FUNCTION_BLOCK "PRG_DSI_Status"
TITLE = Program Status DSI
{ S7_Optimized_Access := 'TRUE' }
AUTHOR : 'A.Schaefer'
VERSION : 0.0
   VAR
      lx_Init { ExternalAccessible := 'False'; ExternalVisible := 'False'; ExternalWritable := 'False'} : Bool;
      lx_Start { ExternalAccessible := 'False'; ExternalVisible := 'False'; ExternalWritable := 'False'} : Bool;
      li_StepCase { ExternalAccessible := 'False'; ExternalVisible := 'False'; ExternalWritable := 'False'} : Int;
      ldt_MQTT { ExternalAccessible := 'False'; ExternalVisible := 'False'; ExternalWritable := 'False'} : Date_And_Time;
      li_Return_LDT { ExternalAccessible := 'False'; ExternalVisible := 'False'; ExternalWritable := 'False'} : Int;
      lfb_R_Trig_Storage {InstructionName := 'R_TRIG'; LibVersion := '1.0'; ExternalAccessible := 'False'; ExternalVisible := 'False'; ExternalWritable := 'False'; S7_SetPoint := 'False'} : R_TRIG;
      lfb_F_Trig_Storage {InstructionName := 'F_TRIG'; LibVersion := '1.0'; ExternalAccessible := 'False'; ExternalVisible := 'False'; ExternalWritable := 'False'; S7_SetPoint := 'False'} : F_TRIG;
      lfb_TON_Status {InstructionName := 'TON_TIME'; LibVersion := '1.0'; ExternalAccessible := 'False'; ExternalVisible := 'False'; ExternalWritable := 'False'; S7_SetPoint := 'False'} : TON_TIME;
      lx_StartStatus { ExternalAccessible := 'False'; ExternalVisible := 'False'; ExternalWritable := 'False'} : Bool;
      lfb_TON_Schritt {InstructionName := 'TON_TIME'; LibVersion := '1.0'; ExternalAccessible := 'False'; ExternalVisible := 'False'; ExternalWritable := 'False'; S7_SetPoint := 'False'} : TON_TIME;
      lx_StartTimer { ExternalAccessible := 'False'; ExternalVisible := 'False'; ExternalWritable := 'False'} : Bool;
   END_VAR


BEGIN
	IF #lx_Init THEN

	    // wait time state
	    #lfb_TON_Status(IN := NOT #lx_StartStatus,
	                    PT := T#2s);

	    // rising/falling edge light barrier DSI
	    #lfb_R_Trig_Storage(CLK := NOT "IX_SSC_LightBarrierStorage_I3");
	    #lfb_F_Trig_Storage(CLK := NOT "IX_SSC_LightBarrierStorage_I3");

	    // state of the DSI transmitted to the cloud
	    IF (#lfb_TON_Status.Q OR #lfb_R_Trig_Storage.Q OR #lfb_F_Trig_Storage.Q) AND NOT #lx_StartStatus THEN
	        #lx_StartStatus := TRUE;
	        #li_Return_LDT := RD_SYS_T(#ldt_MQTT);
	        IF NOT "IX_SSC_LightBarrierStorage_I3" THEN
	            "gtyp_Interface_Dashboard".Subscribe.State_DSI.i_code := 0;
	            "gtyp_Interface_Dashboard".Subscribe.State_DSI.x_active := TRUE;
	        ELSE
	            "gtyp_Interface_Dashboard".Subscribe.State_DSI.i_code := 1;
	            IF #lfb_F_Trig_Storage.Q THEN
	                "gtyp_Interface_Dashboard".Subscribe.State_DSI.x_active := FALSE;
	            END_IF;
	        END_IF;
	        "gtyp_Interface_Dashboard".Subscribe.State_DSI.ldt_ts := DT_TO_LDT(#ldt_MQTT);
	        "gtyp_Interface_Dashboard".Subscribe.State_DSI.s_station := 'dsi';
	        "gtyp_Interface_Dashboard".Subscribe.State_DSI.s_target := '';
	        "gtyp_Interface_Dashboard".Subscribe.State_DSI.s_description := '';
	    END_IF;

	    IF NOT #lfb_TON_Status.Q AND #lx_StartStatus THEN
	        #lx_StartStatus := FALSE;
	    END_IF;
	ELSE
	    #lx_Init := TRUE;
	END_IF;
END_FUNCTION_BLOCK

FUNCTION_BLOCK "PRG_SLD_Ablauf"
TITLE = Program Ablauf SLD
{ S7_Optimized_Access := 'TRUE' }
AUTHOR : 'A.Schaefer'
VERSION : 0.0
   VAR
      lx_Init { ExternalAccessible := 'False'; ExternalVisible := 'False'; ExternalWritable := 'False'} : Bool;
      lx_Start_TON_Wait { ExternalAccessible := 'False'; ExternalVisible := 'False'; ExternalWritable := 'False'} : Bool;
      lx_Time_Error { ExternalAccessible := 'False'; ExternalVisible := 'False'; ExternalWritable := 'False'} : Bool;
      lt_TON_Wait { ExternalAccessible := 'False'; ExternalVisible := 'False'; ExternalWritable := 'False'} : Time;
      lx_Start_TON_State { ExternalAccessible := 'False'; ExternalVisible := 'False'; ExternalWritable := 'False'} : Bool;
      ldt_MQTT { ExternalAccessible := 'False'; ExternalVisible := 'False'; ExternalWritable := 'False'} : Date_And_Time;
      li_Return_LDT { ExternalAccessible := 'False'; ExternalVisible := 'False'; ExternalWritable := 'False'} : Int;
      li_Lights { ExternalAccessible := 'False'; ExternalVisible := 'False'; ExternalWritable := 'False'} : Int;
      li_Lights_old { ExternalAccessible := 'False'; ExternalVisible := 'False'; ExternalWritable := 'False'} : Int;
      lw_ColorValueMin { ExternalAccessible := 'False'; ExternalVisible := 'False'; ExternalWritable := 'False'} : Word;
      li_CounterActual { ExternalAccessible := 'False'; ExternalVisible := 'False'; ExternalWritable := 'False'} : Int;
      lx_White { ExternalAccessible := 'False'; ExternalVisible := 'False'; ExternalWritable := 'False'} : Bool;
      lx_Blue { ExternalAccessible := 'False'; ExternalVisible := 'False'; ExternalWritable := 'False'} : Bool;
      lx_Red { ExternalAccessible := 'False'; ExternalVisible := 'False'; ExternalWritable := 'False'} : Bool;
      li_StepCase { ExternalAccessible := 'False'; ExternalVisible := 'False'; ExternalWritable := 'False'} : Int;
      ls_Color { ExternalAccessible := 'False'; ExternalVisible := 'False'; ExternalWritable := 'False'} : String;
      lfb_TOF_ConveyerBelt_Out {InstructionName := 'TOF_TIME'; LibVersion := '1.0'; ExternalAccessible := 'False'; ExternalVisible := 'False'; ExternalWritable := 'False'; S7_SetPoint := 'False'} : TOF_TIME;
      lfb_TON_Wait {InstructionName := 'TON_TIME'; LibVersion := '1.0'; ExternalAccessible := 'False'; ExternalVisible := 'False'; ExternalWritable := 'False'; S7_SetPoint := 'False'} : TON_TIME;
      lfb_TON_Error {InstructionName := 'TON_TIME'; LibVersion := '1.0'; ExternalAccessible := 'False'; ExternalVisible := 'False'; ExternalWritable := 'False'; S7_SetPoint := 'False'} : TON_TIME;
      lfb_TON_State {InstructionName := 'TON_TIME'; LibVersion := '1.0'; ExternalAccessible := 'False'; ExternalVisible := 'False'; ExternalWritable := 'False'; S7_SetPoint := 'False'} : TON_TIME;
      lfb_F_Trig_Counter {InstructionName := 'F_TRIG'; LibVersion := '1.0'; ExternalAccessible := 'False'; ExternalVisible := 'False'; ExternalWritable := 'False'; S7_SetPoint := 'False'} : F_TRIG;
      lfb_R_Trig_Counter {InstructionName := 'R_TRIG'; LibVersion := '1.0'; ExternalAccessible := 'False'; ExternalVisible := 'False'; ExternalWritable := 'False'; S7_SetPoint := 'False'} : R_TRIG;
   END_VAR


BEGIN
	IF #lx_Init THEN

	    // Restart after set Positioning
	    IF "gtyp_Setup".x_Color_Sensor_Calibration THEN
	        #li_StepCase := 0;
	    END_IF;

	    // wait time state
	    #lfb_TON_State(IN := NOT #lx_Start_TON_State,
	                    PT := T#2s);

	    // state of the SLD cyclically transmitted to the cloud
	    IF (#lfb_TON_State.Q OR (#li_Lights <> #li_Lights_old)) AND NOT #lx_Start_TON_State THEN
	        #li_Lights_old := #li_Lights;
	        #lx_Start_TON_State := TRUE;
	        #li_Return_LDT := RD_SYS_T(#ldt_MQTT);
	        "gtyp_Interface_Dashboard".Subscribe.State_SLD.ldt_ts := DT_TO_LDT(#ldt_MQTT);
	        "gtyp_Interface_Dashboard".Subscribe.State_SLD.i_code := #li_Lights;
	        "gtyp_Interface_Dashboard".Subscribe.State_SLD.s_description := '';
	        "gtyp_Interface_Dashboard".Subscribe.State_SLD.s_station := 'sld';
	        "gtyp_Interface_Dashboard".Subscribe.State_SLD.s_target := '';
	    END_IF;

	    // restart wait time state
	    IF NOT #lfb_TON_State.Q AND #lx_Start_TON_State THEN
	        #lx_Start_TON_State := FALSE;
	    END_IF;

	    // FB TON Wait
	    #lfb_TON_Wait(IN := #lx_Start_TON_Wait,
	                     PT := #lt_TON_Wait);

	    // runtime monitoring error
	    #lfb_TON_Error(IN:= #lx_Time_Error,
	                   PT:= T#30s);

	    // rising edge pulse counter
	    #lfb_R_Trig_Counter(CLK:= "IX_SLD_PulseCounter_I1");

	    // falling edge pulse counter
	    #lfb_F_Trig_Counter(CLK := "IX_SLD_PulseCounter_I1");

	    // step chain SLD
	    CASE #li_StepCase OF

	        0:  // Init
	            #lx_Start_TON_Wait := FALSE;
	            #lx_Time_Error := FALSE;
	            #li_Lights := 1;

	            IF NOT "gtyp_SLD".x_Error AND NOT "gtyp_Setup".x_Color_Sensor_Calibration THEN
	                #li_StepCase := 10;
	            END_IF;

	        10: // turn-on Compressor and wait sequence
	            #li_Lights := 2;
	            "QX_SLD_Compressor_Q2" := TRUE;

	            #lx_Start_TON_Wait := TRUE;
	            #lt_TON_Wait := T#1000ms;

	            IF #lfb_TON_Wait.Q THEN
	                #lx_Start_TON_Wait := FALSE;
	                #li_StepCase := 20;
	            END_IF;

	        20:  // reset Ejectors
	            "QX_SLD_ValveFirstEjectorWhite_Q3"  := FALSE;
	            "QX_SLD_ValveSecondEjectorRed_Q4"   := FALSE;
	            "QX_SLD_ValveThirdEjectorBlue_Q5"   := FALSE;
	            "QX_SLD_M1_ConveyorBelt_Q1"         := FALSE;

	            #lx_Start_TON_Wait := TRUE;
	            #lt_TON_Wait := T#2000ms;

	            IF #lfb_TON_Wait.Q THEN
	                #lx_Start_TON_Wait := FALSE;
	                #li_StepCase := 30;
	            END_IF;

	        30: // turn-off Compressor

	            "QX_SLD_Compressor_Q2" := FALSE;

	            #li_StepCase := 40;

	        40: // start belt if Light barrier I2 active

	            #li_Lights := 1;
	            IF NOT "IX_SLD_LightBarrierInlet_I2" THEN
	                "gtyp_Interface_Dashboard".Subscribe.State_SLD.x_active := TRUE;
	                #li_Lights := 2;
	                "QX_SLD_Compressor_Q2"      := TRUE;
	                "QX_SLD_M1_ConveyorBelt_Q1" := TRUE;
	                #lw_ColorValueMin           := 40000;
	                #li_CounterActual := 0;
	                #lx_Blue := FALSE;
	                #lx_Red := FALSE;
	                #lx_White := FALSE;
	                #li_StepCase := 50;
	            END_IF;

	        50: // take the min Value of the Color sensor
	            IF #lw_ColorValueMin > "IW_SLD_ColorSensor_A4" THEN
	                #lw_ColorValueMin := "IW_SLD_ColorSensor_A4";
	            END_IF;

	            #lx_Time_Error := TRUE;

	            // Stop when light barrier I3 on
	            IF NOT "IX_SLD_LightBarrierBehindColorSensor_I3" THEN
	                #lx_Time_Error  := FALSE;
	                #li_StepCase    := 60;
	            END_IF;

	            // runtime error
	            IF #lfb_TON_Error.Q THEN
	                #li_Lights                  := 4;
	                #lx_Time_Error              := FALSE;
	                "QX_SLD_Compressor_Q2"      := FALSE;
	                "QX_SLD_M1_ConveyorBelt_Q1" := FALSE;
	                "gtyp_Interface_Dashboard".Subscribe.State_SLD.x_active := FALSE;
	                "gtyp_SLD".x_Error          := TRUE;
	                #li_StepCase                := 0;
	            END_IF;

	        60: // analyze color

	            IF #lw_ColorValueMin >= "gtyp_SLD".w_Threshold_Red_Blue THEN
	                #lx_Blue := TRUE;
	            ELSIF #lw_ColorValueMin <= "gtyp_SLD".w_Threshold_White_Red THEN
	                #lx_White := TRUE;
	            ELSIF #lw_ColorValueMin > "gtyp_SLD".w_Threshold_White_Red AND #lw_ColorValueMin < "gtyp_SLD".w_Threshold_Red_Blue THEN
	                #lx_Red := TRUE;
	            END_IF;

	            // actual counter
	            IF #lfb_R_Trig_Counter.Q OR #lfb_F_Trig_Counter.Q THEN
	                #li_CounterActual := #li_CounterActual + 1;
	            END_IF;

	            // Reached counter value and color set Ejector
	            IF (#li_CounterActual = "gtyp_SLD".i_CounterValue_Blue) AND #lx_Blue THEN
	                "QX_SLD_ValveThirdEjectorBlue_Q5" := TRUE;
	                #li_Return_LDT := RD_SYS_T(#ldt_MQTT);
	                "gtyp_SLD".Workpiece.s_state := 'PROCESSED';
	                "gtyp_SLD".History[7].i_code := 700;
	                "gtyp_SLD".History[7].ldt_ts := DT_TO_LDT(#ldt_MQTT);
	                #li_StepCase := 70;
	            ELSIF (#li_CounterActual = "gtyp_SLD".i_CounterValue_White) AND #lx_White THEN
	                "QX_SLD_ValveFirstEjectorWhite_Q3" := TRUE;
	                #li_Return_LDT := RD_SYS_T(#ldt_MQTT);
	                "gtyp_SLD".Workpiece.s_state := 'PROCESSED';
	                "gtyp_SLD".History[7].i_code := 700;
	                "gtyp_SLD".History[7].ldt_ts := DT_TO_LDT(#ldt_MQTT);
	                #li_StepCase := 70;
	            ELSIF (#li_CounterActual = "gtyp_SLD".i_CounterValue_Red) AND #lx_Red THEN
	                "QX_SLD_ValveSecondEjectorRed_Q4" := TRUE;
	                #li_Return_LDT := RD_SYS_T(#ldt_MQTT);
	                "gtyp_SLD".Workpiece.s_state := 'PROCESSED';
	                "gtyp_SLD".History[7].i_code := 700;
	                "gtyp_SLD".History[7].ldt_ts := DT_TO_LDT(#ldt_MQTT);
	                #li_StepCase := 70;
	            ELSIF (#li_CounterActual = 80) THEN
	                #li_Lights := 4;
	                "gtyp_SLD".x_Error := TRUE;
	                #li_StepCase := 70;
	            END_IF;

	        70: // wait sequence
	            #lx_Start_TON_Wait := TRUE;
	            #lt_TON_Wait := T#500ms;

	            IF #lfb_TON_Wait.Q THEN
	                "QX_SLD_ValveThirdEjectorBlue_Q5" := FALSE;
	                "QX_SLD_ValveFirstEjectorWhite_Q3" := FALSE;
	                "QX_SLD_ValveSecondEjectorRed_Q4" := FALSE;
	                #lx_Start_TON_Wait := FALSE;
	                #li_StepCase := 80;
	            END_IF;

	        80: // wait sequence

	            #lx_Start_TON_Wait := TRUE;
	            #lt_TON_Wait := T#2000ms;

	            IF #lfb_TON_Wait.Q THEN
	                "QX_SLD_Compressor_Q2" := FALSE;
	                #lx_Start_TON_Wait := FALSE;
	                #li_StepCase := 90;
	            END_IF;

	        90: // Stop belt
	            "QX_SLD_M1_ConveyorBelt_Q1"    := FALSE;
	            #li_StepCase := 40;
	        // Statement section ELSE
	        ELSE
	            ;
	    END_CASE;

	ELSE
	    "gtyp_SLD".x_Error := FALSE;
	    #li_Lights := 1;
	    #lx_Init := TRUE;
	END_IF;
END_FUNCTION_BLOCK

FUNCTION_BLOCK "PRG_HBW_Axis_Horizontal"
TITLE = Program Axis horizontal HBW
{ S7_Optimized_Access := 'TRUE' }
AUTHOR : 'A.Schaefer'
VERSION : 0.0
   VAR
      lx_Init { ExternalAccessible := 'False'; ExternalVisible := 'False'; ExternalWritable := 'False'} : Bool;
      lfb_Horizontal_Axis { ExternalAccessible := 'False'; ExternalVisible := 'False'; ExternalWritable := 'False'; S7_SetPoint := 'False'} : "FB_Axis";
   END_VAR


BEGIN
	IF #lx_Init THEN

	    // FB Axis horizontal
	    #lfb_Horizontal_Axis(ini_Axis               := 6,
	                         indi_Increment          := "gtyp_HBW".Horizontal_Axis.di_Increment,
	                         inx_Ref_Switch         := "IX_HBW_RefSwitchHorizontalAxis_I1",
	                         inx_Referencing        := "gtyp_HBW".Horizontal_Axis.x_Reference,
	                         inx_Start_Positioning  := "gtyp_HBW".Horizontal_Axis.x_Start_Positioning,
	                         indi_Target_Position   := "gtyp_HBW".Horizontal_Axis.di_Target_Position,
	                         ini_PWM                := "gtyp_HBW".Horizontal_Axis.i_PWM,
	                         inouttyp_Config        := "gtyp_HBW".Horizontal_Axis.Config,
	                         inouttyp_Setup         := "gtyp_SetupAxis");

	    "QX_HBW_M2_HorizontalTowardsRack_Q3"            := #lfb_Horizontal_Axis.outx_Motor_Pos;
	    "QX_HBW_M2_HorizontalTowardsConveyorBelt_Q4"    := #lfb_Horizontal_Axis.outx_Motor_Neg;
	    "QW_HBW_PWM_HorizontalAxis_M2"                  := #lfb_Horizontal_Axis.outi_Motor_PWM;
	    "gtyp_HBW".Horizontal_Axis.di_Actual_Position   := #lfb_Horizontal_Axis.outdi_Actual_Position;
	    "gtyp_HBW".Horizontal_Axis.x_Referenced         := #lfb_Horizontal_Axis.outx_Referenced;
	    "gtyp_HBW".Horizontal_Axis.x_Position_Reached   := #lfb_Horizontal_Axis.outx_Position_Reached;
	ELSE
	    #lx_Init := TRUE;
	END_IF;
END_FUNCTION_BLOCK

FUNCTION_BLOCK "PRG_SSC_Light"
TITLE = Program Lights
{ S7_Optimized_Access := 'TRUE' }
AUTHOR : 'A.Schaefer'
VERSION : 0.0
   VAR
      lx_Init { ExternalAccessible := 'False'; ExternalVisible := 'False'; ExternalWritable := 'False'} : Bool;
      lx_Start { ExternalAccessible := 'False'; ExternalVisible := 'False'; ExternalWritable := 'False'} : Bool;
      li_StepCase { ExternalAccessible := 'False'; ExternalVisible := 'False'; ExternalWritable := 'False'} : Int;
      ldt_MQTT { ExternalAccessible := 'False'; ExternalVisible := 'False'; ExternalWritable := 'False'} : Date_And_Time;
      lldt_ts_old { ExternalAccessible := 'False'; ExternalVisible := 'False'; ExternalWritable := 'False'} : LDT;
      li_Return_LDT { ExternalAccessible := 'False'; ExternalVisible := 'False'; ExternalWritable := 'False'} : Int;
      lfb_TOF_Camera {InstructionName := 'TOF_TIME'; LibVersion := '1.0'; ExternalAccessible := 'False'; ExternalVisible := 'False'; ExternalWritable := 'False'; S7_SetPoint := 'False'} : TOF_TIME;
      lfb_TON_Schritt {InstructionName := 'TON_TIME'; LibVersion := '1.0'; ExternalAccessible := 'False'; ExternalVisible := 'False'; ExternalWritable := 'False'; S7_SetPoint := 'False'} : TON_TIME;
      lfb_blinker_cam { ExternalAccessible := 'False'; ExternalVisible := 'False'; ExternalWritable := 'False'; S7_SetPoint := 'False'} : "FB_Blinker";
      lfb_blinker_config { ExternalAccessible := 'False'; ExternalVisible := 'False'; ExternalWritable := 'False'; S7_SetPoint := 'False'} : "FB_Blinker";
      lx_StartTimer { ExternalAccessible := 'False'; ExternalVisible := 'False'; ExternalWritable := 'False'} : Bool;
   END_VAR


BEGIN
	IF #lx_Init THEN

	    // if camera sen picture - Red light flash
	    IF "gtyp_Interface_Dashboard".Subscribe.CameraPicture.ldt_ts > #lldt_ts_old THEN
	        #lldt_ts_old := "gtyp_Interface_Dashboard".Subscribe.CameraPicture.ldt_ts;
	        #lfb_blinker_cam(int_periodendauer := T#50ms);
	    END_IF;

	    // reload flash
	    "QX_SSC_LED_Red_Online_Q8":= #lfb_blinker_cam.outx_blinker;

	    // FB flash config
	    #lfb_blinker_config(int_periodendauer := T#500ms);

	    //  Deciding which state
	    //  Setup - Calibration State
	    IF "gtyp_Setup".x_Set_Pos_Activ OR "gtyp_Setup".x_Color_Sensor_Calibration
	                                    OR "gtyp_Setup".x_Counter_Value_Calibration
	                                    OR "gtyp_Setup".x_Clean_Rack_HBW THEN
	        "QX_SSC_LED_Green_Q5"  := #lfb_blinker_config.outx_blinker;
	        "QX_SSC_LED_Yellow_Q6" := #lfb_blinker_config.outx_blinker;
	        "QX_SSC_LED_Red_Q7"    := #lfb_blinker_config.outx_blinker;
	    //  Error State
	    ELSIF ("gtyp_Interface_Dashboard".Subscribe.State_HBW.i_code = 4)
	        OR ("gtyp_Interface_Dashboard".Subscribe.State_MPO.i_code = 4)
	        OR ("gtyp_Interface_Dashboard".Subscribe.State_SLD.i_code = 4)
	        OR ("gtyp_Interface_Dashboard".Subscribe.State_VGR.i_code = 4) THEN
	        "QX_SSC_LED_Green_Q5" := FALSE;
	        "QX_SSC_LED_Yellow_Q6" := FALSE;
	        "QX_SSC_LED_Red_Q7" := TRUE;
	    //  Proccessing State
	    ELSIF ("gtyp_Interface_Dashboard".Subscribe.State_HBW.i_code = 2)
	        OR ("gtyp_Interface_Dashboard".Subscribe.State_MPO.i_code = 2)
	        OR ("gtyp_Interface_Dashboard".Subscribe.State_SLD.i_code = 2)
	        OR ("gtyp_Interface_Dashboard".Subscribe.State_VGR.i_code = 2) THEN
	            "QX_SSC_LED_Green_Q5" := FALSE;
	            "QX_SSC_LED_Yellow_Q6" := TRUE;
	            "QX_SSC_LED_Red_Q7" := FALSE;
	    //  Idle State
	    ELSIF ("gtyp_Interface_Dashboard".Subscribe.State_HBW.i_code = 1)
	        AND ("gtyp_Interface_Dashboard".Subscribe.State_MPO.i_code = 1)
	        AND ("gtyp_Interface_Dashboard".Subscribe.State_SLD.i_code = 1)
	        AND ("gtyp_Interface_Dashboard".Subscribe.State_VGR.i_code = 1) THEN
	            "QX_SSC_LED_Green_Q5" := TRUE;
	            "QX_SSC_LED_Yellow_Q6" := FALSE;
	            "QX_SSC_LED_Red_Q7" := FALSE;
	    //  nothing State
	    ELSE
	        "QX_SSC_LED_Green_Q5" := FALSE;
	        "QX_SSC_LED_Yellow_Q6" := FALSE;
	        "QX_SSC_LED_Red_Q7" := FALSE;
	    END_IF;


	ELSE
	    #lx_Init := TRUE;
	END_IF;
END_FUNCTION_BLOCK

FUNCTION_BLOCK "PRG_DSO_Status"
TITLE = Program Status DSO
{ S7_Optimized_Access := 'TRUE' }
AUTHOR : 'A.Schaefer'
VERSION : 0.0
   VAR
      lx_Init { ExternalAccessible := 'False'; ExternalVisible := 'False'; ExternalWritable := 'False'} : Bool;
      lx_Start { ExternalAccessible := 'False'; ExternalVisible := 'False'; ExternalWritable := 'False'} : Bool;
      li_StepCase { ExternalAccessible := 'False'; ExternalVisible := 'False'; ExternalWritable := 'False'} : Int;
      ldt_MQTT { ExternalAccessible := 'False'; ExternalVisible := 'False'; ExternalWritable := 'False'} : Date_And_Time;
      li_Return_LDT { ExternalAccessible := 'False'; ExternalVisible := 'False'; ExternalWritable := 'False'} : Int;
      li_code_old { ExternalAccessible := 'False'; ExternalVisible := 'False'; ExternalWritable := 'False'} : Int;
      lfb_R_Trig_Outsourcing {InstructionName := 'R_TRIG'; LibVersion := '1.0'; ExternalAccessible := 'False'; ExternalVisible := 'False'; ExternalWritable := 'False'; S7_SetPoint := 'False'} : R_TRIG;
      lfb_R_Trig_Take_Workpiece {InstructionName := 'R_TRIG'; LibVersion := '1.0'; ExternalAccessible := 'False'; ExternalVisible := 'False'; ExternalWritable := 'False'; S7_SetPoint := 'False'} : R_TRIG;
      lfb_TON_Status {InstructionName := 'TON_TIME'; LibVersion := '1.0'; ExternalAccessible := 'False'; ExternalVisible := 'False'; ExternalWritable := 'False'; S7_SetPoint := 'False'} : TON_TIME;
      lfb_TON_End_Order {InstructionName := 'TON_TIME'; LibVersion := '1.0'; ExternalAccessible := 'False'; ExternalVisible := 'False'; ExternalWritable := 'False'; S7_SetPoint := 'False'} : TON_TIME;
      lx_StartStatus { ExternalAccessible := 'False'; ExternalVisible := 'False'; ExternalWritable := 'False'} : Bool;
      lx_StartEndOrder { ExternalAccessible := 'False'; ExternalVisible := 'False'; ExternalWritable := 'False'} : Bool;
      lx_StartTimer { ExternalAccessible := 'False'; ExternalVisible := 'False'; ExternalWritable := 'False'} : Bool;
   END_VAR


BEGIN
	IF #lx_Init THEN

	    // wait time state
	    #lfb_TON_Status(IN := NOT #lx_StartStatus,
	                    PT := T#2s);

	    // rising/falling edge light barrier DSI
	    #lfb_R_Trig_Outsourcing(CLK := NOT "IX_SSC_LightBarrierOutsourcing_I4");
	    #lfb_R_Trig_Take_Workpiece(CLK := "IX_SSC_LightBarrierOutsourcing_I4");

	    // start wait time end order
	    IF NOT "IX_SSC_LightBarrierOutsourcing_I4" AND ("gtyp_Interface_Dashboard".Subscribe.State_Order.s_state = 'SHIPPED') THEN
	        #lx_StartEndOrder := TRUE;
	    END_IF;

	    // wait time end order
	    #lfb_TON_End_Order(IN := #lx_StartEndOrder,
	                       PT := T#5s);

	    IF #lfb_R_Trig_Take_Workpiece.Q OR #lfb_TON_End_Order.Q THEN
	        #lx_StartEndOrder := FALSE;
	        "gtyp_Interface_Dashboard".Subscribe.State_Order.ldt_ts := DT_TO_LDT(#ldt_MQTT);
	        "gtyp_Interface_Dashboard".Subscribe.State_Order.s_state := 'WAITING_FOR_ORDER';
	        "gtyp_Interface_Dashboard".Subscribe.State_Order.s_type := '';
	        "gtyp_Interface_Dashboard".Subscribe.State_DSO.x_active := FALSE;
	    END_IF;

	    // state of the DSO transmitted to the cloud
	    IF (#lfb_TON_Status.Q OR #lfb_R_Trig_Outsourcing.Q OR #lfb_R_Trig_Take_Workpiece.Q) AND NOT #lx_StartStatus THEN
	        #lx_StartStatus := TRUE;
	        #li_Return_LDT := RD_SYS_T(#ldt_MQTT);
	        IF NOT "IX_SSC_LightBarrierOutsourcing_I4" THEN
	            "gtyp_Interface_Dashboard".Subscribe.State_DSO.i_code := 0;
	        ELSE
	            "gtyp_Interface_Dashboard".Subscribe.State_DSO.i_code := 1;
	        END_IF;
	        "gtyp_Interface_Dashboard".Subscribe.State_DSO.ldt_ts := DT_TO_LDT(#ldt_MQTT);
	        "gtyp_Interface_Dashboard".Subscribe.State_DSO.s_station := 'dso';
	        "gtyp_Interface_Dashboard".Subscribe.State_DSO.s_target := '';
	        "gtyp_Interface_Dashboard".Subscribe.State_DSO.s_description := '';
	    END_IF;

	    IF NOT #lfb_TON_Status.Q AND #lx_StartStatus THEN
	        #lx_StartStatus := FALSE;
	    END_IF;
	ELSE
	    #lx_Init := TRUE;
	    #lx_StartEndOrder := FALSE;
	END_IF;
END_FUNCTION_BLOCK

FUNCTION_BLOCK "PRG_SSC_Set_Positioning"
TITLE = Program Set Positioning SSC
{ S7_Optimized_Access := 'TRUE' }
AUTHOR : 'A.Schaefer'
VERSION : 0.0
   VAR
      lx_Init { ExternalAccessible := 'False'; ExternalVisible := 'False'; ExternalWritable := 'False'} : Bool;
      lx_Start_TON_Wait { ExternalAccessible := 'False'; ExternalVisible := 'False'; ExternalWritable := 'False'} : Bool;
      lx_Start_Positioning_m { ExternalAccessible := 'False'; ExternalVisible := 'False'; ExternalWritable := 'False'} : Bool;
      lt_TON_Wait { ExternalAccessible := 'False'; ExternalVisible := 'False'; ExternalWritable := 'False'} : Time;
      li_StepCase { ExternalAccessible := 'False'; ExternalVisible := 'False'; ExternalWritable := 'False'} : Int;
      ldi_Pos_Horizontal { ExternalAccessible := 'False'; ExternalVisible := 'False'; ExternalWritable := 'False'} : DInt;
      ldi_Pos_Vertical { ExternalAccessible := 'False'; ExternalVisible := 'False'; ExternalWritable := 'False'} : DInt;
      lfb_R_Trig_Deaktivate {InstructionName := 'R_TRIG'; LibVersion := '1.0'; ExternalAccessible := 'False'; ExternalVisible := 'False'; ExternalWritable := 'False'; S7_SetPoint := 'False'} : R_TRIG;
      lfb_TON_Wait {InstructionName := 'TON_TIME'; LibVersion := '1.0'; ExternalAccessible := 'False'; ExternalVisible := 'False'; ExternalWritable := 'False'; S7_SetPoint := 'False'} : TON_TIME;
   END_VAR


BEGIN
	IF #lx_Init THEN

	    // FB TON Wait
	    #lfb_TON_Wait(IN := #lx_Start_TON_Wait,
	                  PT := #lt_TON_Wait);

	    #lfb_R_Trig_Deaktivate(CLK:= NOT "gtyp_Setup".x_Set_Pos_Activ
	                           OR NOT (("gtyp_Setup".i_Pos_Selection > 0)
	                           AND ("gtyp_Setup".i_Pos_Selection < 21)));
	    // Deaktivate step 10
	    IF #lfb_R_Trig_Deaktivate.Q THEN
	        "gtyp_SSC".Horizontal_Axis.x_Start_Positioning := FALSE;
	        "gtyp_SSC".Vertical_Axis.x_Start_Positioning := FALSE;
	        "gtyp_SSC".Horizontal_Axis.x_Reference := FALSE;
	        "gtyp_SSC".Vertical_Axis.x_Reference := FALSE;
	        "gtyp_Setup".x_Start_Positioning := FALSE;
	        "gtyp_Setup".x_Final_Positioning := FALSE;
	        "gtyp_Setup".x_Home_Positioning := FALSE;
	        "gtyp_Setup".x_Start_Offset := FALSE;
	        #lx_Start_Positioning_m := FALSE;
	        IF (#li_StepCase > 10) THEN
	            #li_StepCase            := 70;
	        END_IF;
	    END_IF;

	    // Set Positioning activ?
	    IF "gtyp_Setup".x_Set_Pos_Activ
	        AND (("gtyp_Setup".i_Pos_Selection > 0)
	        AND ("gtyp_Setup".i_Pos_Selection < 21))
	        AND ((#li_StepCase = 40)
	        OR (#li_StepCase = 60)) THEN

	        // Deciding which Position
	        // Position - Centre
	        IF "gtyp_Setup".i_Pos_Selection = 1 THEN
	            #ldi_Pos_Horizontal := "gtyp_SSC".di_Pos_Centre_Horizontal;
	            #ldi_Pos_Vertical := "gtyp_SSC".di_Pos_Centre_Vertical;
	            // Position - HBW
	        ELSIF "gtyp_Setup".i_Pos_Selection = 2 THEN
	            #ldi_Pos_Horizontal := "gtyp_SSC".di_Pos_HBW_Horizontal;
	            #ldi_Pos_Vertical := "gtyp_SSC".di_Pos_HBW_Vertical;
	        END_IF;
	    END_IF;

	    // Set Positioning activ?
	    IF NOT "gtyp_Setup".x_Set_Pos_Activ THEN
	        "gtyp_Setup".i_Pos_Selection := 0;
	    END_IF;

	    // step chain HBW
	    CASE #li_StepCase OF

	        0:  // init
	            #lx_Start_TON_Wait := FALSE;
	            #li_StepCase := 10;

	        10:  // Set Positioning activ?
	            IF "gtyp_Setup".x_Set_Pos_Activ
	                AND (("gtyp_Setup".i_Pos_Selection > 0)
	                AND ("gtyp_Setup".i_Pos_Selection < 21)) THEN
	                "gtyp_SSC".Horizontal_Axis.x_Start_Positioning := FALSE;
	                "gtyp_SSC".Vertical_Axis.x_Start_Positioning := FALSE;
	                "gtyp_SSC".Horizontal_Axis.x_Reference := FALSE;
	                "gtyp_SSC".Vertical_Axis.x_Reference := FALSE;
	                "gtyp_Setup".x_Start_Positioning := FALSE;
	                "gtyp_Setup".x_Final_Positioning := FALSE;
	                "gtyp_Setup".x_Home_Positioning  := FALSE;
	                "gtyp_Setup".x_Start_Offset := FALSE;
	                #li_StepCase := 20;
	            END_IF;

	        20: //homing vertical/horizontal axis

	            "gtyp_SSC".Horizontal_Axis.x_Reference := TRUE;
	            "gtyp_SSC".Vertical_Axis.x_Reference := TRUE;

	            IF NOT "gtyp_SSC".Horizontal_Axis.x_Referenced AND NOT "gtyp_SSC".Vertical_Axis.x_Referenced THEN
	                #li_StepCase := 30;
	            END_IF;

	        30: // homed vertical/horizontal axis
	            IF "gtyp_SSC".Horizontal_Axis.x_Referenced THEN
	                "gtyp_SSC".Horizontal_Axis.x_Reference := FALSE;
	            END_IF;
	            IF "gtyp_SSC".Vertical_Axis.x_Referenced THEN
	                "gtyp_SSC".Vertical_Axis.x_Reference := FALSE;
	            END_IF;

	            IF "gtyp_SSC".Horizontal_Axis.x_Referenced AND "gtyp_SSC".Vertical_Axis.x_Referenced THEN
	                "gtyp_SSC".Horizontal_Axis.x_Reference := FALSE;
	                "gtyp_SSC".Vertical_Axis.x_Reference := FALSE;
	                #li_StepCase := 40;
	            END_IF;

	        40:  // Start Positioning Step next
	            IF "gtyp_Setup".x_Start_Positioning OR #lx_Start_Positioning_m THEN
	                #lx_Start_Positioning_m := FALSE;
	                #li_StepCase            := 50;
	            END_IF;

	        50: // Position vertical/horizontal HBW
	            "gtyp_SSC".Horizontal_Axis.di_Target_Position := #ldi_Pos_Horizontal;
	            "gtyp_SSC".Horizontal_Axis.x_Start_Positioning := TRUE;
	            "gtyp_SSC".Vertical_Axis.di_Target_Position := #ldi_Pos_Vertical;
	            "gtyp_SSC".Vertical_Axis.x_Start_Positioning := TRUE;

	            IF ("gtyp_SSC".Horizontal_Axis.di_Actual_Position <= (#ldi_Pos_Horizontal + "gtyp_SSC".Horizontal_Axis.Config.di_Pos_Window))
	                AND ("gtyp_SSC".Horizontal_Axis.di_Actual_Position >= (#ldi_Pos_Horizontal - "gtyp_SSC".Horizontal_Axis.Config.di_Pos_Window))
	                AND "gtyp_SSC".Horizontal_Axis.x_Position_Reached THEN
	                "gtyp_SSC".Horizontal_Axis.x_Start_Positioning := FALSE;
	            END_IF;

	            IF ("gtyp_SSC".Vertical_Axis.di_Actual_Position <= (#ldi_Pos_Vertical + "gtyp_SSC".Vertical_Axis.Config.di_Pos_Window))
	                AND ("gtyp_SSC".Vertical_Axis.di_Actual_Position >= (#ldi_Pos_Vertical - "gtyp_SSC".Vertical_Axis.Config.di_Pos_Window))
	                AND "gtyp_SSC".Vertical_Axis.x_Position_Reached THEN
	                "gtyp_SSC".Vertical_Axis.x_Start_Positioning := FALSE;
	            END_IF;

	            IF ("gtyp_SSC".Horizontal_Axis.di_Actual_Position <= (#ldi_Pos_Horizontal + "gtyp_SSC".Horizontal_Axis.Config.di_Pos_Window))
	                AND ("gtyp_SSC".Horizontal_Axis.di_Actual_Position >= (#ldi_Pos_Horizontal - "gtyp_SSC".Horizontal_Axis.Config.di_Pos_Window))
	                AND "gtyp_SSC".Horizontal_Axis.x_Position_Reached
	                AND ("gtyp_SSC".Vertical_Axis.di_Actual_Position <= (#ldi_Pos_Vertical + "gtyp_SSC".Vertical_Axis.Config.di_Pos_Window))
	                AND ("gtyp_SSC".Vertical_Axis.di_Actual_Position >= (#ldi_Pos_Vertical - "gtyp_SSC".Vertical_Axis.Config.di_Pos_Window))
	                AND "gtyp_SSC".Vertical_Axis.x_Position_Reached THEN
	                "gtyp_SSC".Horizontal_Axis.x_Start_Positioning := FALSE;
	                "gtyp_SSC".Vertical_Axis.x_Start_Positioning := FALSE;
	                "gtyp_Setup".x_Start_Positioning := FALSE;
	                #li_StepCase := 60;
	            END_IF;

	        60: // Deciding which doing

	            // Start new Positioning
	            IF "gtyp_Setup".x_Start_Positioning OR "gtyp_Setup".x_Home_Positioning THEN
	                #lx_Start_Positioning_m := TRUE;
	                #li_StepCase            := 10;
	            ELSIF #lfb_R_Trig_Deaktivate.Q THEN
	                "gtyp_Setup".x_Home_Positioning := FALSE;
	                #li_StepCase                    := 70;
	            END_IF;

	        70: //homing vertical/horizontal axis

	            "gtyp_SSC".Horizontal_Axis.x_Reference := TRUE;
	            "gtyp_SSC".Vertical_Axis.x_Reference := TRUE;

	            IF NOT "gtyp_SSC".Horizontal_Axis.x_Referenced AND NOT "gtyp_SSC".Vertical_Axis.x_Referenced THEN
	                #li_StepCase := 80;
	            END_IF;

	        80: // homed vertical/horizontal axis
	            IF "gtyp_SSC".Horizontal_Axis.x_Referenced THEN
	                "gtyp_SSC".Horizontal_Axis.x_Reference := FALSE;
	            END_IF;
	            IF "gtyp_SSC".Vertical_Axis.x_Referenced THEN
	                "gtyp_SSC".Vertical_Axis.x_Reference := FALSE;
	            END_IF;

	            IF "gtyp_SSC".Horizontal_Axis.x_Referenced AND "gtyp_SSC".Vertical_Axis.x_Referenced THEN
	                "gtyp_SSC".Horizontal_Axis.x_Reference := FALSE;
	                "gtyp_SSC".Vertical_Axis.x_Reference := FALSE;
	                #li_StepCase := 0;
	            END_IF;

	            // Statement section ELSE
	        ELSE
	            ;
	    END_CASE;

	    IF (("gtyp_Setup".i_Pos_Selection > 0)
	        AND ("gtyp_Setup".i_Pos_Selection < 21)) THEN
	        // Reload Pos Value
	        "gtyp_Setup".di_Pos_Horizontal := #ldi_Pos_Horizontal;
	        "gtyp_Setup".di_Pos_Vertical := #ldi_Pos_Vertical;
	        "gtyp_Setup".di_Pos_Rotate := 0;
	    END_IF;
	ELSE
	    #lx_Init := TRUE;
	END_IF;
END_FUNCTION_BLOCK

FUNCTION_BLOCK "PRG_HBW_Set_Positioning"
TITLE = Program Set Positioning HBW
{ S7_Optimized_Access := 'TRUE' }
AUTHOR : 'A.Schaefer'
VERSION : 0.0
   VAR
      lx_Init { ExternalAccessible := 'False'; ExternalVisible := 'False'; ExternalWritable := 'False'} : Bool;
      lx_Start_TON_Wait { ExternalAccessible := 'False'; ExternalVisible := 'False'; ExternalWritable := 'False'} : Bool;
      lx_Start_Positioning_m { ExternalAccessible := 'False'; ExternalVisible := 'False'; ExternalWritable := 'False'} : Bool;
      lx_Start_FinalPositioning_m { ExternalAccessible := 'False'; ExternalVisible := 'False'; ExternalWritable := 'False'} : Bool;
      lx_Start_Offset_m { ExternalAccessible := 'False'; ExternalVisible := 'False'; ExternalWritable := 'False'} : Bool;
      lt_TON_Wait { ExternalAccessible := 'False'; ExternalVisible := 'False'; ExternalWritable := 'False'} : Time;
      li_Counter_Hor { ExternalAccessible := 'False'; ExternalVisible := 'False'; ExternalWritable := 'False'} : Int;
      li_Counter_Ver { ExternalAccessible := 'False'; ExternalVisible := 'False'; ExternalWritable := 'False'} : Int;
      li_Counter_Act_Hor { ExternalAccessible := 'False'; ExternalVisible := 'False'; ExternalWritable := 'False'} : Int;
      li_Counter_Act_Ver { ExternalAccessible := 'False'; ExternalVisible := 'False'; ExternalWritable := 'False'} : Int;
      li_Counter { ExternalAccessible := 'False'; ExternalVisible := 'False'; ExternalWritable := 'False'} : Int;
      li_StepCase { ExternalAccessible := 'False'; ExternalVisible := 'False'; ExternalWritable := 'False'} : Int;
      ldi_Pos_Horizontal { ExternalAccessible := 'False'; ExternalVisible := 'False'; ExternalWritable := 'False'} : DInt;
      ldi_Pos_Vertical { ExternalAccessible := 'False'; ExternalVisible := 'False'; ExternalWritable := 'False'} : DInt;
      ldi_Offset_Vertical { ExternalAccessible := 'False'; ExternalVisible := 'False'; ExternalWritable := 'False'} : DInt;
      lfb_R_Trig_Deaktivate {InstructionName := 'R_TRIG'; LibVersion := '1.0'; ExternalAccessible := 'False'; ExternalVisible := 'False'; ExternalWritable := 'False'; S7_SetPoint := 'False'} : R_TRIG;
      lfb_TON_Wait {InstructionName := 'TON_TIME'; LibVersion := '1.0'; ExternalAccessible := 'False'; ExternalVisible := 'False'; ExternalWritable := 'False'; S7_SetPoint := 'False'} : TON_TIME;
   END_VAR


BEGIN
	IF #lx_Init THEN

	    // FB TON Wait
	    #lfb_TON_Wait(IN := #lx_Start_TON_Wait,
	                  PT := #lt_TON_Wait);

	    #lfb_R_Trig_Deaktivate(CLK:= NOT "gtyp_Setup".x_Set_Pos_Activ
	                           OR NOT (("gtyp_Setup".i_Pos_Selection > 20)
	                           AND ("gtyp_Setup".i_Pos_Selection < 41)));
	    // Deaktivate step 110
	    IF #lfb_R_Trig_Deaktivate.Q THEN
	        "gtyp_HBW".Horizontal_Axis.x_Start_Positioning := FALSE;
	        "gtyp_HBW".Vertical_Axis.x_Start_Positioning := FALSE;
	        "gtyp_HBW".Horizontal_Axis.x_Reference := FALSE;
	        "gtyp_HBW".Vertical_Axis.x_Reference := FALSE;
	        "gtyp_Setup".x_Start_Positioning := FALSE;
	        "gtyp_Setup".x_Final_Positioning := FALSE;
	        "gtyp_Setup".x_Home_Positioning := FALSE;
	        "gtyp_Setup".x_Start_Offset := FALSE;
	        "QX_HBW_M4_CantileverBackward_Q8" := FALSE;
	        "QX_HBW_M4_CantileverForward_Q7" := FALSE;
	        IF (#li_StepCase > 10) THEN
	            #li_StepCase := 110;
	        END_IF;
	    END_IF;

	    // Set Positioning activ?
	    IF "gtyp_Setup".x_Set_Pos_Activ
	        AND (("gtyp_Setup".i_Pos_Selection > 20)
	        AND ("gtyp_Setup".i_Pos_Selection < 41))
	        AND ((#li_StepCase = 40)
	        OR (#li_StepCase = 60)
	        OR (#li_StepCase = 80)
	        OR (#li_StepCase = 100)) THEN

	        // Deciding which Position
	        // Position - Belt
	        IF "gtyp_Setup".i_Pos_Selection = 21 THEN
	            #ldi_Pos_Horizontal := "gtyp_HBW".di_PosBelt_Horizontal;
	            #ldi_Pos_Vertical := "gtyp_HBW".di_PosBelt_Vertical;
	            #ldi_Offset_Vertical := "gtyp_HBW".di_Offset_Pos_Belt_Vertical;
	            // Position - A1
	        ELSIF "gtyp_Setup".i_Pos_Selection = 22 THEN
	            #ldi_Pos_Horizontal := "gtyp_HBW".di_PosRack_A1_Horizontal;
	            #ldi_Pos_Vertical := "gtyp_HBW".di_PosRack_A1_Vertical;
	            #ldi_Offset_Vertical := "gtyp_HBW".di_Offset_Pos_Rack_Vertical;
	            // Position - B2
	        ELSIF "gtyp_Setup".i_Pos_Selection = 23 THEN
	            #ldi_Pos_Horizontal := "gtyp_HBW".di_PosRack_B2_Horizontal;
	            #ldi_Pos_Vertical := "gtyp_HBW".di_PosRack_B2_Vertical;
	            #ldi_Offset_Vertical := "gtyp_HBW".di_Offset_Pos_Rack_Vertical;
	            // Position - C3
	        ELSIF "gtyp_Setup".i_Pos_Selection = 24 THEN
	            #ldi_Pos_Horizontal := "gtyp_HBW".di_PosRack_C3_Horizontal;
	            #ldi_Pos_Vertical := "gtyp_HBW".di_PosRack_C3_Vertical;
	            #ldi_Offset_Vertical := "gtyp_HBW".di_Offset_Pos_Rack_Vertical;
	        END_IF;
	    END_IF;

	    // Set Positioning activ?
	    IF NOT "gtyp_Setup".x_Set_Pos_Activ THEN
	        "gtyp_Setup".i_Pos_Selection := 0;
	    END_IF;

	    // step chain HBW
	    CASE #li_StepCase OF

	        0:  // init
	            #lx_Start_TON_Wait := FALSE;
	            #li_StepCase := 10;

	        10:  // Set Positioning activ?
	            IF "gtyp_Setup".x_Set_Pos_Activ
	                AND (("gtyp_Setup".i_Pos_Selection > 20)
	                AND ("gtyp_Setup".i_Pos_Selection < 41)) THEN

	                "gtyp_HBW".Horizontal_Axis.x_Start_Positioning  := FALSE;
	                "gtyp_HBW".Vertical_Axis.x_Start_Positioning    := FALSE;
	                "gtyp_HBW".Horizontal_Axis.x_Reference          := FALSE;
	                "gtyp_HBW".Vertical_Axis.x_Reference            := FALSE;
	                "gtyp_Setup".x_Start_Positioning            := FALSE;
	                "gtyp_Setup".x_Final_Positioning            := FALSE;
	                "gtyp_Setup".x_Home_Positioning             := FALSE;
	                "gtyp_Setup".x_Start_Offset                 := FALSE;
	                "QX_HBW_M4_CantileverBackward_Q8"               := FALSE;
	                "QX_HBW_M4_CantileverForward_Q7"                := FALSE;
	                #li_StepCase                                    := 20;
	            END_IF;

	        20: //homing vertical/horizontal axis

	            "gtyp_HBW".Horizontal_Axis.x_Reference := TRUE;
	            "gtyp_HBW".Vertical_Axis.x_Reference := TRUE;

	            IF NOT "gtyp_HBW".Horizontal_Axis.x_Referenced AND NOT "gtyp_HBW".Vertical_Axis.x_Referenced THEN
	                #li_StepCase := 30;
	            END_IF;

	        30: // homed vertical/horizontal axis
	            IF "gtyp_HBW".Horizontal_Axis.x_Referenced THEN
	                "gtyp_HBW".Horizontal_Axis.x_Reference := FALSE;
	            END_IF;
	            IF "gtyp_HBW".Vertical_Axis.x_Referenced THEN
	                "gtyp_HBW".Vertical_Axis.x_Reference := FALSE;
	            END_IF;

	            IF "gtyp_HBW".Horizontal_Axis.x_Referenced AND "gtyp_HBW".Vertical_Axis.x_Referenced THEN
	                "gtyp_HBW".Horizontal_Axis.x_Reference := FALSE;
	                "gtyp_HBW".Vertical_Axis.x_Reference := FALSE;
	                #li_StepCase := 40;
	            END_IF;

	        40: // Start Positioning Step next
	            IF "gtyp_Setup".x_Start_Positioning OR #lx_Start_Positioning_m OR #lx_Start_FinalPositioning_m OR #lx_Start_Offset_m THEN
	                #lx_Start_Positioning_m := FALSE;
	                #li_StepCase := 50;
	            END_IF;

	        50: // Position vertical/horizontal HBW
	            "gtyp_HBW".Horizontal_Axis.di_Target_Position   := #ldi_Pos_Horizontal;
	            "gtyp_HBW".Horizontal_Axis.x_Start_Positioning  := TRUE;
	            "gtyp_HBW".Vertical_Axis.di_Target_Position     := #ldi_Pos_Vertical;
	            "gtyp_HBW".Vertical_Axis.x_Start_Positioning    := TRUE;

	            IF ("gtyp_HBW".Horizontal_Axis.di_Actual_Position <= (#ldi_Pos_Horizontal + "gtyp_HBW".Horizontal_Axis.Config.di_Pos_Window))
	                AND ("gtyp_HBW".Horizontal_Axis.di_Actual_Position >= (#ldi_Pos_Horizontal - "gtyp_HBW".Horizontal_Axis.Config.di_Pos_Window))
	                AND "gtyp_HBW".Horizontal_Axis.x_Position_Reached THEN
	                "gtyp_HBW".Horizontal_Axis.x_Start_Positioning := FALSE;
	            END_IF;

	            IF ("gtyp_HBW".Vertical_Axis.di_Actual_Position <= (#ldi_Pos_Vertical + "gtyp_HBW".Vertical_Axis.Config.di_Pos_Window))
	                AND ("gtyp_HBW".Vertical_Axis.di_Actual_Position >= (#ldi_Pos_Vertical - "gtyp_HBW".Vertical_Axis.Config.di_Pos_Window))
	                AND "gtyp_HBW".Vertical_Axis.x_Position_Reached THEN
	                "gtyp_HBW".Vertical_Axis.x_Start_Positioning := FALSE;
	            END_IF;

	            IF ("gtyp_HBW".Horizontal_Axis.di_Actual_Position <= (#ldi_Pos_Horizontal + "gtyp_HBW".Horizontal_Axis.Config.di_Pos_Window))
	                AND ("gtyp_HBW".Horizontal_Axis.di_Actual_Position >= (#ldi_Pos_Horizontal - "gtyp_HBW".Horizontal_Axis.Config.di_Pos_Window))
	                AND "gtyp_HBW".Horizontal_Axis.x_Position_Reached
	                AND ("gtyp_HBW".Vertical_Axis.di_Actual_Position <= (#ldi_Pos_Vertical + "gtyp_HBW".Vertical_Axis.Config.di_Pos_Window))
	                AND ("gtyp_HBW".Vertical_Axis.di_Actual_Position >= (#ldi_Pos_Vertical - "gtyp_HBW".Vertical_Axis.Config.di_Pos_Window))
	                AND "gtyp_HBW".Vertical_Axis.x_Position_Reached THEN
	                "gtyp_HBW".Horizontal_Axis.x_Start_Positioning  := FALSE;
	                "gtyp_HBW".Vertical_Axis.x_Start_Positioning    := FALSE;
	                "gtyp_Setup".x_Start_Positioning          := FALSE;
	                #li_StepCase := 60;
	            END_IF;

	        60: // Deciding which doing

	            // Start new Positioning
	            IF "gtyp_Setup".x_Start_Positioning THEN
	                #lx_Start_Positioning_m := TRUE;
	                #li_StepCase := 10;
	            // Start Final Positioning
	            ELSIF "gtyp_Setup".x_Final_Positioning OR #lx_Start_FinalPositioning_m OR #lx_Start_Offset_m THEN
	                #lx_Start_FinalPositioning_m := FALSE;
	                #li_StepCase := 70;
	            // Deaktivate Set Positioning
	            ELSIF #lfb_R_Trig_Deaktivate.Q OR "gtyp_Setup".x_Home_Positioning THEN
	                "gtyp_Setup".x_Home_Positioning := FALSE;
	                #li_StepCase := 110;
	            END_IF;

	        70: // Final Positioning - Cantilever Forward

	            "QX_HBW_M4_CantileverBackward_Q8" := FALSE;
	            "QX_HBW_M4_CantileverForward_Q7" := TRUE;

	            IF "IX_HBW_SwitchCantileverFront_I5" AND NOT "IX_HBW_SwitchCantileverBack_I6" THEN
	                "QX_HBW_M4_CantileverBackward_Q8" := FALSE;
	                "QX_HBW_M4_CantileverForward_Q7" := FALSE;
	                "gtyp_Setup".x_Final_Positioning := FALSE;
	                #li_StepCase := 80;
	            END_IF;

	        80: // Deciding which doing

	            // Start new Positioning
	            IF "gtyp_Setup".x_Start_Positioning THEN
	                #lx_Start_Positioning_m := TRUE;
	                #li_StepCase := 110;
	                // Start Final Positioning
	            ELSIF "gtyp_Setup".x_Final_Positioning THEN
	                #lx_Start_FinalPositioning_m := TRUE;
	                #li_StepCase := 110;
	                // Start Final Positioning
	            ELSIF "gtyp_Setup".x_Start_Offset OR #lx_Start_Offset_m THEN
	                #lx_Start_Offset_m := FALSE;
	                #li_StepCase := 90;
	                // Deaktivate Set Positioning
	            ELSIF #lfb_R_Trig_Deaktivate.Q OR "gtyp_Setup".x_Home_Positioning THEN
	                "gtyp_Setup".x_Home_Positioning := FALSE;
	                #li_StepCase := 110;
	            END_IF;

	        90: // Position vertical+offset HBW
	            "gtyp_HBW".Vertical_Axis.di_Target_Position := #ldi_Pos_Vertical - #ldi_Offset_Vertical;
	            "gtyp_HBW".Vertical_Axis.x_Start_Positioning := TRUE;

	            IF ("gtyp_HBW".Vertical_Axis.di_Actual_Position <= (#ldi_Pos_Vertical - #ldi_Offset_Vertical + "gtyp_HBW".Vertical_Axis.Config.di_Pos_Window))
	                AND ("gtyp_HBW".Vertical_Axis.di_Actual_Position >= (#ldi_Pos_Vertical - #ldi_Offset_Vertical - "gtyp_HBW".Vertical_Axis.Config.di_Pos_Window))
	                AND "gtyp_HBW".Vertical_Axis.x_Position_Reached THEN
	                "gtyp_HBW".Vertical_Axis.x_Start_Positioning := FALSE;
	                "gtyp_Setup".x_Start_Offset            := FALSE;
	                #li_StepCase := 100;
	            END_IF;

	        100: // Deciding which doing

	            // Start new Positioning
	            IF "gtyp_Setup".x_Start_Positioning THEN
	                #lx_Start_Positioning_m := TRUE;
	                #li_StepCase := 110;
	                // Start Final Positioning
	            ELSIF "gtyp_Setup".x_Final_Positioning THEN
	                #lx_Start_FinalPositioning_m := TRUE;
	                #li_StepCase := 110;
	                // Start Final Positioning
	            ELSIF "gtyp_Setup".x_Start_Offset THEN
	                #lx_Start_Offset_m := true;
	                #li_StepCase := 110;
	                // Deaktivate Set Positioning
	            ELSIF #lfb_R_Trig_Deaktivate.Q OR "gtyp_Setup".x_Home_Positioning THEN
	                "gtyp_Setup".x_Home_Positioning := FALSE;
	                #li_StepCase := 110;
	            END_IF;

	        110: // Position vertical HBW
	            "gtyp_HBW".Vertical_Axis.di_Target_Position := #ldi_Pos_Vertical;
	            "gtyp_HBW".Vertical_Axis.x_Start_Positioning := TRUE;

	            IF ("gtyp_HBW".Vertical_Axis.di_Actual_Position <= (#ldi_Pos_Vertical + "gtyp_HBW".Vertical_Axis.Config.di_Pos_Window))
	                AND ("gtyp_HBW".Vertical_Axis.di_Actual_Position >= (#ldi_Pos_Vertical - "gtyp_HBW".Vertical_Axis.Config.di_Pos_Window))
	                AND "gtyp_HBW".Vertical_Axis.x_Position_Reached THEN
	                "gtyp_HBW".Vertical_Axis.x_Start_Positioning := FALSE;
	                #li_StepCase := 120;
	            END_IF;

	        120: // Position vertical Back HBW

	            "QX_HBW_M4_CantileverBackward_Q8" := TRUE;
	            "QX_HBW_M4_CantileverForward_Q7" := FALSE;

	            IF NOT "IX_HBW_SwitchCantileverFront_I5" AND "IX_HBW_SwitchCantileverBack_I6" THEN
	                "QX_HBW_M4_CantileverBackward_Q8" := FALSE;
	                "QX_HBW_M4_CantileverForward_Q7" := FALSE;
	                #li_StepCase := 130;
	            END_IF;

	        130: // homing vertical/horizontal axis

	            "gtyp_HBW".Horizontal_Axis.x_Reference := TRUE;
	            "gtyp_HBW".Vertical_Axis.x_Reference := TRUE;

	            IF NOT "gtyp_HBW".Horizontal_Axis.x_Referenced AND NOT "gtyp_HBW".Vertical_Axis.x_Referenced THEN
	                #li_StepCase := 140;
	            END_IF;

	        140: //homed vertical/horizontal axis
	            IF "gtyp_HBW".Horizontal_Axis.x_Referenced THEN
	                "gtyp_HBW".Horizontal_Axis.x_Reference := FALSE;
	            END_IF;
	            IF "gtyp_HBW".Vertical_Axis.x_Referenced THEN
	                "gtyp_HBW".Vertical_Axis.x_Reference := FALSE;
	            END_IF;

	            IF "gtyp_HBW".Horizontal_Axis.x_Referenced AND "gtyp_HBW".Vertical_Axis.x_Referenced THEN
	                "gtyp_HBW".Horizontal_Axis.x_Reference := FALSE;
	                "gtyp_HBW".Vertical_Axis.x_Reference := FALSE;
	                #li_StepCase := 0;
	            END_IF;

	    // Statement section ELSE
	    ELSE
	        ;
	    END_CASE;

	    IF (("gtyp_Setup".i_Pos_Selection > 20)
	        AND ("gtyp_Setup".i_Pos_Selection < 41)) THEN
	        // Reload Pos Value
	        "gtyp_Setup".di_Pos_Horizontal := #ldi_Pos_Horizontal;
	        "gtyp_Setup".di_Pos_Vertical := #ldi_Pos_Vertical;
	        "gtyp_Setup".di_Pos_Rotate := 0;
	    END_IF;
	ELSE
	    #lx_Init := TRUE;
	END_IF;
END_FUNCTION_BLOCK

FUNCTION_BLOCK "PRG_VGR_Set_Positioning"
TITLE = Program Set Positioning VGR
{ S7_Optimized_Access := 'TRUE' }
AUTHOR : 'A.Schaefer'
VERSION : 0.0
   VAR
      lx_Init { ExternalAccessible := 'False'; ExternalVisible := 'False'; ExternalWritable := 'False'} : Bool;
      lx_Start_TON_Wait { ExternalAccessible := 'False'; ExternalVisible := 'False'; ExternalWritable := 'False'} : Bool;
      lx_Start_Positioning_m { ExternalAccessible := 'False'; ExternalVisible := 'False'; ExternalWritable := 'False'} : Bool;
      lx_Start_FinalPositioning_m { ExternalAccessible := 'False'; ExternalVisible := 'False'; ExternalWritable := 'False'} : Bool;
      lx_Start_TON_State { ExternalAccessible := 'False'; ExternalVisible := 'False'; ExternalWritable := 'False'} : Bool;
      lt_TON_Wait { ExternalAccessible := 'False'; ExternalVisible := 'False'; ExternalWritable := 'False'} : Time;
      ldt_MQTT { ExternalAccessible := 'False'; ExternalVisible := 'False'; ExternalWritable := 'False'} : Date_And_Time;
      li_Return_LDT { ExternalAccessible := 'False'; ExternalVisible := 'False'; ExternalWritable := 'False'} : Int;
      li_Lights { ExternalAccessible := 'False'; ExternalVisible := 'False'; ExternalWritable := 'False'} : Int;
      li_Lights_old { ExternalAccessible := 'False'; ExternalVisible := 'False'; ExternalWritable := 'False'} : Int;
      lx_State_activ { ExternalAccessible := 'False'; ExternalVisible := 'False'; ExternalWritable := 'False'} : Bool;
      li_StepCase { ExternalAccessible := 'False'; ExternalVisible := 'False'; ExternalWritable := 'False'} : Int;
      li_Counter { ExternalAccessible := 'False'; ExternalVisible := 'False'; ExternalWritable := 'False'} : Int;
      ldi_Pos_SLD_X { ExternalAccessible := 'False'; ExternalVisible := 'False'; ExternalWritable := 'False'} : DInt;
      ldi_Pos_SLD_Y { ExternalAccessible := 'False'; ExternalVisible := 'False'; ExternalWritable := 'False'} : DInt;
      ldi_Pos_SLD_Z { ExternalAccessible := 'False'; ExternalVisible := 'False'; ExternalWritable := 'False'} : DInt;
      ldi_Pos_Horizontal { ExternalAccessible := 'False'; ExternalVisible := 'False'; ExternalWritable := 'False'} : DInt;
      ldi_Pos_Vertical { ExternalAccessible := 'False'; ExternalVisible := 'False'; ExternalWritable := 'False'} : DInt;
      ldi_Pos_Rotate { ExternalAccessible := 'False'; ExternalVisible := 'False'; ExternalWritable := 'False'} : DInt;
      ldi_Offset_Vertical { ExternalAccessible := 'False'; ExternalVisible := 'False'; ExternalWritable := 'False'} : DInt;
      ls_Color { ExternalAccessible := 'False'; ExternalVisible := 'False'; ExternalWritable := 'False'} : String;
      ls_Target { ExternalAccessible := 'False'; ExternalVisible := 'False'; ExternalWritable := 'False'} : String;
      lfb_TON_Wait {InstructionName := 'TON_TIME'; LibVersion := '1.0'; ExternalAccessible := 'False'; ExternalVisible := 'False'; ExternalWritable := 'False'; S7_SetPoint := 'False'} : TON_TIME;
      lfb_TON_State {InstructionName := 'TON_TIME'; LibVersion := '1.0'; ExternalAccessible := 'False'; ExternalVisible := 'False'; ExternalWritable := 'False'; S7_SetPoint := 'False'} : TON_TIME;
      lfb_R_Trig_Deaktivate {InstructionName := 'R_TRIG'; LibVersion := '1.0'; ExternalAccessible := 'False'; ExternalVisible := 'False'; ExternalWritable := 'False'; S7_SetPoint := 'False'} : R_TRIG;
      lfb_R_Trig_NiO {InstructionName := 'R_TRIG'; LibVersion := '1.0'; ExternalAccessible := 'False'; ExternalVisible := 'False'; ExternalWritable := 'False'; S7_SetPoint := 'False'} : R_TRIG;
   END_VAR


BEGIN
	IF #lx_Init THEN

	    // FB TON Wait
	    #lfb_TON_Wait(IN := #lx_Start_TON_Wait,
	                  PT := #lt_TON_Wait);

	    #lfb_R_Trig_Deaktivate(CLK := NOT "gtyp_Setup".x_Set_Pos_Activ
	                           OR NOT (("gtyp_Setup".i_Pos_Selection > 40)
	                           AND ("gtyp_Setup".i_Pos_Selection < 61)));
	    // Deaktivate step 150
	    IF #lfb_R_Trig_Deaktivate.Q THEN
	        "gtyp_VGR".horizontal_Axis.x_Start_Positioning := FALSE;
	        "gtyp_VGR".vertical_Axis.x_Start_Positioning := FALSE;
	        "gtyp_VGR".rotate_Axis.x_Start_Positioning := FALSE;
	        "gtyp_VGR".horizontal_Axis.x_Reference := FALSE;
	        "gtyp_VGR".vertical_Axis.x_Reference := FALSE;
	        "gtyp_VGR".rotate_Axis.x_Reference := FALSE;
	        "gtyp_Setup".x_Start_Positioning := FALSE;
	        "gtyp_Setup".x_Final_Positioning := FALSE;
	        "gtyp_Setup".x_Home_Positioning := FALSE;
	        "gtyp_Setup".x_Start_Offset := FALSE;
	        IF (#li_StepCase > 10) THEN
	            #li_StepCase := 150;
	        END_IF;
	    END_IF;

	    // Set Positioning activ?
	    IF "gtyp_Setup".x_Set_Pos_Activ
	        AND (("gtyp_Setup".i_Pos_Selection > 40)
	        AND ("gtyp_Setup".i_Pos_Selection < 61))
	        AND ((#li_StepCase = 80)
	        OR (#li_StepCase = 120)
	        OR (#li_StepCase = 140)) THEN

	        // Deciding which Position
	        // Position - Color
	        IF "gtyp_Setup".i_Pos_Selection = 41 THEN
	            #ldi_Pos_Horizontal := "gtyp_VGR".di_Pos_Color_horizontal;
	            #ldi_Pos_Vertical := "gtyp_VGR".di_Pos_Color_vertical;
	            #ldi_Pos_Rotate := "gtyp_VGR".di_Pos_Color_rotate;
	            #ldi_Offset_Vertical := "gtyp_VGR".di_Offset_Pos_DSI_NFC_vertical;
	            // Position - DSI Collect
	        ELSIF "gtyp_Setup".i_Pos_Selection = 42 THEN
	            #ldi_Pos_Horizontal := "gtyp_VGR".di_Pos_DSI_horizontal;
	            #ldi_Pos_Vertical := "gtyp_VGR".di_Pos_DSI_Collect_vertical;
	            #ldi_Pos_Rotate := "gtyp_VGR".di_Pos_DSI_rotate;
	            #ldi_Offset_Vertical := "gtyp_VGR".di_Offset_Pos_DSI_NFC_vertical;
	            // Position - DSI Discard
	        ELSIF "gtyp_Setup".i_Pos_Selection = 43 THEN
	            #ldi_Pos_Horizontal := "gtyp_VGR".di_Pos_DSI_horizontal;
	            #ldi_Pos_Vertical := "gtyp_VGR".di_Pos_DSI_Discard_vertical;
	            #ldi_Pos_Rotate := "gtyp_VGR".di_Pos_DSI_rotate;
	            #ldi_Offset_Vertical := "gtyp_VGR".di_Offset_Pos_DSI_NFC_vertical;
	            // Position - DSO Collect
	        ELSIF "gtyp_Setup".i_Pos_Selection = 44 THEN
	            #ldi_Pos_Horizontal := "gtyp_VGR".di_Pos_DSO_horizontal;
	            #ldi_Pos_Vertical := "gtyp_VGR".di_Pos_DSO_Collect_vertical;
	            #ldi_Pos_Rotate := "gtyp_VGR".di_Pos_DSO_rotate;
	            #ldi_Offset_Vertical := "gtyp_VGR".di_Offset_Pos_DSO_vertical;
	            // Position - DSO Discard
	        ELSIF "gtyp_Setup".i_Pos_Selection = 45 THEN
	            #ldi_Pos_Horizontal := "gtyp_VGR".di_Pos_DSO_horizontal;
	            #ldi_Pos_Vertical := "gtyp_VGR".di_Pos_DSO_Discard_vertical;
	            #ldi_Pos_Rotate := "gtyp_VGR".di_Pos_DSO_rotate;
	            #ldi_Offset_Vertical := "gtyp_VGR".di_Offset_Pos_DSO_vertical;
	            // Position - HBW Collect
	        ELSIF "gtyp_Setup".i_Pos_Selection = 46 THEN
	            #ldi_Pos_Horizontal := "gtyp_VGR".di_Pos_HBW_horizontal;
	            #ldi_Pos_Vertical := "gtyp_VGR".di_Pos_HBW_Collect_vertical;
	            #ldi_Pos_Rotate := "gtyp_VGR".di_Pos_HBW_rotate;
	            #ldi_Offset_Vertical := "gtyp_VGR".di_Offset_Pos_HBW_vertical;
	            // Position - HBW Discard
	        ELSIF "gtyp_Setup".i_Pos_Selection = 47 THEN
	            #ldi_Pos_Horizontal := "gtyp_VGR".di_Pos_HBW_horizontal;
	            #ldi_Pos_Vertical := "gtyp_VGR".di_Pos_HBW_Discard_vertical;
	            #ldi_Pos_Rotate := "gtyp_VGR".di_Pos_HBW_rotate;
	            #ldi_Offset_Vertical := "gtyp_VGR".di_Offset_Pos_HBW_vertical;
	            // Position - MPO
	        ELSIF "gtyp_Setup".i_Pos_Selection = 48 THEN
	            #ldi_Pos_Horizontal := "gtyp_VGR".di_Pos_MPO_horizontal;
	            #ldi_Pos_Vertical := "gtyp_VGR".di_Pos_MPO_vertical;
	            #ldi_Pos_Rotate := "gtyp_VGR".di_Pos_MPO_rotate;
	            #ldi_Offset_Vertical := "gtyp_VGR".di_Offset_Pos_MPO_vertical;
	            // Position - NFC
	        ELSIF "gtyp_Setup".i_Pos_Selection = 49 THEN
	            #ldi_Pos_Horizontal := "gtyp_VGR".di_Pos_NFC_horizontal;
	            #ldi_Pos_Vertical := "gtyp_VGR".di_Pos_NFC_vertical;
	            #ldi_Pos_Rotate := "gtyp_VGR".di_Pos_NFC_rotate;
	            #ldi_Offset_Vertical := "gtyp_VGR".di_Offset_Pos_DSI_NFC_vertical;
	            // Position - NiO
	        ELSIF "gtyp_Setup".i_Pos_Selection = 50 THEN
	            #ldi_Pos_Horizontal := "gtyp_VGR".di_Pos_NiO_horizontal;
	            #ldi_Pos_Vertical := "gtyp_VGR".di_Pos_NiO_vertical;
	            #ldi_Pos_Rotate := "gtyp_VGR".di_Pos_NiO_rotate;
	            #ldi_Offset_Vertical := 500;
	            // Position - SLD Blue
	        ELSIF "gtyp_Setup".i_Pos_Selection = 51 THEN
	            #ldi_Pos_Horizontal := "gtyp_VGR".di_Pos_SLD_Blue_horizontal;
	            #ldi_Pos_Vertical := "gtyp_VGR".di_Pos_SLD_Blue_vertical;
	            #ldi_Pos_Rotate := "gtyp_VGR".di_Pos_SLD_Blue_rotate;
	            #ldi_Offset_Vertical := 500;
	            // Position - SLD Red
	        ELSIF "gtyp_Setup".i_Pos_Selection = 52 THEN
	            #ldi_Pos_Horizontal := "gtyp_VGR".di_Pos_SLD_Red_horizontal;
	            #ldi_Pos_Vertical := "gtyp_VGR".di_Pos_SLD_Red_vertical;
	            #ldi_Pos_Rotate := "gtyp_VGR".di_Pos_SLD_Red_rotate;
	            #ldi_Offset_Vertical := 500;
	            // Position - SLD White
	        ELSIF "gtyp_Setup".i_Pos_Selection = 53 THEN
	            #ldi_Pos_Horizontal := "gtyp_VGR".di_Pos_SLD_White_horizontal;
	            #ldi_Pos_Vertical := "gtyp_VGR".di_Pos_SLD_White_vertical;
	            #ldi_Pos_Rotate := "gtyp_VGR".di_Pos_SLD_White_rotate;
	            #ldi_Offset_Vertical := 500;
	        END_IF;
	    END_IF;

	    // Set Positioning activ?
	    IF NOT "gtyp_Setup".x_Set_Pos_Activ THEN
	        "gtyp_Setup".i_Pos_Selection := 0;
	    END_IF;

	        // step chain HBW
	    CASE #li_StepCase OF

	        0:  // init
	            #lx_Start_TON_Wait := FALSE;
	            #li_StepCase := 10;

	        10:  // Set Positioning activ?
	            IF "gtyp_Setup".x_Set_Pos_Activ
	                AND (("gtyp_Setup".i_Pos_Selection > 40)
	                AND ("gtyp_Setup".i_Pos_Selection < 61)) THEN

	                "gtyp_VGR".horizontal_Axis.x_Start_Positioning := FALSE;
	                "gtyp_VGR".vertical_Axis.x_Start_Positioning := FALSE;
	                "gtyp_VGR".rotate_Axis.x_Start_Positioning := FALSE;
	                "gtyp_VGR".horizontal_Axis.x_Reference := FALSE;
	                "gtyp_VGR".vertical_Axis.x_Reference := FALSE;
	                "gtyp_VGR".rotate_Axis.x_Reference := FALSE;
	                "gtyp_Setup".x_Start_Positioning := FALSE;
	                "gtyp_Setup".x_Final_Positioning := FALSE;
	                "gtyp_Setup".x_Home_Positioning := FALSE;
	                "gtyp_Setup".x_Start_Offset := FALSE;
	                "gtyp_VGR".vertical_Axis.i_PWM := 800;
	                #li_StepCase := 20;
	            END_IF;

	        20: // homing vertical axis
	            "gtyp_VGR".vertical_Axis.x_Reference := TRUE;

	            IF NOT "gtyp_VGR".vertical_Axis.x_Referenced THEN
	                #li_StepCase := 30;
	            END_IF;

	        30: // homed vertical axis
	            IF "gtyp_VGR".vertical_Axis.x_Referenced THEN
	                "gtyp_VGR".vertical_Axis.x_Reference := FALSE;
	                #li_StepCase := 40;
	            END_IF;

	        40: // homing horizontal axis
	            "gtyp_VGR".horizontal_Axis.x_Reference := TRUE;

	            IF NOT "gtyp_VGR".horizontal_Axis.x_Referenced THEN
	                #li_StepCase := 50;
	            END_IF;

	        50: // homed horizontal axis
	            IF "gtyp_VGR".horizontal_Axis.x_Referenced THEN
	                "gtyp_VGR".horizontal_Axis.x_Reference := FALSE;
	                #li_StepCase := 60;
	            END_IF;

	        60: // homing rotate axis
	            "gtyp_VGR".rotate_Axis.x_Reference := TRUE;

	            IF NOT "gtyp_VGR".rotate_Axis.x_Referenced THEN
	                #li_StepCase := 70;
	            END_IF;

	        70: // homed rotate axis
	            IF "gtyp_VGR".rotate_Axis.x_Referenced THEN
	                "gtyp_VGR".rotate_Axis.x_Reference := FALSE;
	                #li_StepCase := 80;
	            END_IF;

	        80:  // Start Positioning Step next
	            IF "gtyp_Setup".x_Start_Positioning OR #lx_Start_Positioning_m OR #lx_Start_FinalPositioning_m THEN
	                #lx_Start_Positioning_m := FALSE;
	                #li_StepCase := 90;
	            END_IF;

	        90: // Position rotate Axis
	            "gtyp_VGR".rotate_Axis.di_Target_Position   := #ldi_Pos_Rotate;
	            "gtyp_VGR".rotate_Axis.x_Start_Positioning  := TRUE;

	            IF ("gtyp_VGR".rotate_Axis.di_Actual_Position <= (#ldi_Pos_Rotate + "gtyp_VGR".rotate_Axis.Config.di_Pos_Window))
	                AND ("gtyp_VGR".rotate_Axis.di_Actual_Position >= (#ldi_Pos_Rotate - "gtyp_VGR".rotate_Axis.Config.di_Pos_Window))
	                AND "gtyp_VGR".rotate_Axis.x_Position_Reached THEN
	                "gtyp_VGR".rotate_Axis.x_Start_Positioning := FALSE;
	                #li_StepCase := 100;
	            END_IF;

	        100: // Position horizontal Axis
	            "gtyp_VGR".horizontal_Axis.di_Target_Position := #ldi_Pos_Horizontal;
	            "gtyp_VGR".horizontal_Axis.x_Start_Positioning := TRUE;

	            IF ("gtyp_VGR".horizontal_Axis.di_Actual_Position <= (#ldi_Pos_Horizontal + "gtyp_VGR".horizontal_Axis.Config.di_Pos_Window))
	                AND ("gtyp_VGR".horizontal_Axis.di_Actual_Position >= (#ldi_Pos_Horizontal - "gtyp_VGR".horizontal_Axis.Config.di_Pos_Window))
	                AND "gtyp_VGR".horizontal_Axis.x_Position_Reached THEN
	                "gtyp_VGR".horizontal_Axis.x_Start_Positioning := FALSE;
	                #li_StepCase := 110;
	            END_IF;

	        110: // Position vertical Axis + Offset
	            "gtyp_VGR".vertical_Axis.i_PWM := 500;
	            "gtyp_VGR".vertical_Axis.di_Target_Position := #ldi_Pos_Vertical - #ldi_Offset_Vertical;
	            "gtyp_VGR".vertical_Axis.x_Start_Positioning := TRUE;

	            IF ("gtyp_VGR".vertical_Axis.di_Actual_Position <= (#ldi_Pos_Vertical - #ldi_Offset_Vertical + "gtyp_VGR".vertical_Axis.Config.di_Pos_Window))
	                AND ("gtyp_VGR".vertical_Axis.di_Actual_Position >= (#ldi_Pos_Vertical - #ldi_Offset_Vertical - "gtyp_VGR".vertical_Axis.Config.di_Pos_Window))
	                AND "gtyp_VGR".vertical_Axis.x_Position_Reached THEN
	                "gtyp_VGR".vertical_Axis.x_Start_Positioning := FALSE;
	                "gtyp_Setup".x_Start_Positioning := FALSE;
	                #li_StepCase := 120;
	            END_IF;

	        120: // Deciding which doing

	            // Start new Positioning
	            IF "gtyp_Setup".x_Start_Positioning THEN
	                #lx_Start_Positioning_m := TRUE;
	                #li_StepCase := 10;
	                // Start Final Positioning
	            ELSIF "gtyp_Setup".x_Final_Positioning OR #lx_Start_FinalPositioning_m THEN
	                #lx_Start_FinalPositioning_m := FALSE;
	                #li_StepCase := 130;
	                // Deaktivate Set Positioning
	            ELSIF #lfb_R_Trig_Deaktivate.Q OR "gtyp_Setup".x_Home_Positioning THEN
	                "gtyp_Setup".x_Home_Positioning := FALSE;
	                #li_StepCase := 150;
	            END_IF;

	        130: // Position vertical Axis
	            "gtyp_VGR".vertical_Axis.di_Target_Position := #ldi_Pos_Vertical;
	            "gtyp_VGR".vertical_Axis.x_Start_Positioning := TRUE;

	            IF ("gtyp_VGR".vertical_Axis.di_Actual_Position <= (#ldi_Pos_Vertical + "gtyp_VGR".vertical_Axis.Config.di_Pos_Window))
	                AND ("gtyp_VGR".vertical_Axis.di_Actual_Position >= (#ldi_Pos_Vertical - "gtyp_VGR".vertical_Axis.Config.di_Pos_Window))
	                AND "gtyp_VGR".vertical_Axis.x_Position_Reached THEN
	                "gtyp_VGR".vertical_Axis.x_Start_Positioning := FALSE;
	                "gtyp_Setup".x_Final_Positioning := FALSE;
	                #li_StepCase := 140;
	            END_IF;

	        140: // Deciding which doing

	            // Start new Positioning
	            IF "gtyp_Setup".x_Start_Positioning THEN
	                #lx_Start_Positioning_m := TRUE;
	                #li_StepCase := 10;
	                // Start Final Positioning
	            ELSIF "gtyp_Setup".x_Final_Positioning THEN
	                #lx_Start_FinalPositioning_m := TRUE;
	                #li_StepCase := 10;
	                // Start Final Positioning
	            ELSIF #lfb_R_Trig_Deaktivate.Q OR "gtyp_Setup".x_Home_Positioning THEN
	                "gtyp_Setup".x_Home_Positioning := FALSE;
	                #li_StepCase := 150;
	            END_IF;

	        150: // homing vertical axis
	            "gtyp_VGR".vertical_Axis.i_PWM := 800;
	            "gtyp_VGR".vertical_Axis.x_Reference := TRUE;

	            IF NOT "gtyp_VGR".vertical_Axis.x_Referenced THEN
	                #li_StepCase := 160;
	            END_IF;

	        160: // homed vertical axis
	            IF "gtyp_VGR".vertical_Axis.x_Referenced THEN
	                "gtyp_VGR".vertical_Axis.x_Reference := FALSE;
	                #li_StepCase := 170;
	            END_IF;

	        170: // homing horizontal axis
	            "gtyp_VGR".horizontal_Axis.x_Reference := TRUE;

	            IF NOT "gtyp_VGR".horizontal_Axis.x_Referenced THEN
	                #li_StepCase := 180;
	            END_IF;

	        180: // homed horizontal axis
	            IF "gtyp_VGR".horizontal_Axis.x_Referenced THEN
	                "gtyp_VGR".horizontal_Axis.x_Reference := FALSE;
	                #li_StepCase := 0;
	            END_IF;

	            // Statement section ELSE
	        ELSE
	            ;
	    END_CASE;

	    IF (("gtyp_Setup".i_Pos_Selection > 40)
	        AND ("gtyp_Setup".i_Pos_Selection < 61)) THEN
	        // Reload Pos Value
	        "gtyp_Setup".di_Pos_Horizontal := #ldi_Pos_Horizontal;
	        "gtyp_Setup".di_Pos_Vertical := #ldi_Pos_Vertical;
	        "gtyp_Setup".di_Pos_Rotate := #ldi_Pos_Rotate;
	    END_IF;
	ELSE
	    #lx_Init := TRUE;
	END_IF;
END_FUNCTION_BLOCK

FUNCTION_BLOCK "PRG_SSC_Ablauf"
TITLE = Program Ablauf SSC
{ S7_Optimized_Access := 'TRUE' }
AUTHOR : 'A.Schaefer'
VERSION : 0.0
   VAR
      lx_Init { ExternalAccessible := 'False'; ExternalVisible := 'False'; ExternalWritable := 'False'} : Bool;
      lx_FirstCentre { ExternalAccessible := 'False'; ExternalVisible := 'False'; ExternalWritable := 'False'} : Bool;
      lx_Start { ExternalAccessible := 'False'; ExternalVisible := 'False'; ExternalWritable := 'False'} : Bool;
      lx_Start_TON_State { ExternalAccessible := 'False'; ExternalVisible := 'False'; ExternalWritable := 'False'} : Bool;
      lt_TON_Wait { ExternalAccessible := 'False'; ExternalVisible := 'False'; ExternalWritable := 'False'} : Time;
      li_StepCase { ExternalAccessible := 'False'; ExternalVisible := 'False'; ExternalWritable := 'False'} : Int;
      ldi_TargetPosition_Horizontal { ExternalAccessible := 'False'; ExternalVisible := 'False'; ExternalWritable := 'False'} : DInt;
      ldi_TargetPosition_Vertical { ExternalAccessible := 'False'; ExternalVisible := 'False'; ExternalWritable := 'False'} : DInt;
      lldt_ts_old { ExternalAccessible := 'False'; ExternalVisible := 'False'; ExternalWritable := 'False'} : LDT;
      ldt_write { ExternalAccessible := 'False'; ExternalVisible := 'False'; ExternalWritable := 'False'} : Date_And_Time;
      li_Return_write { ExternalAccessible := 'False'; ExternalVisible := 'False'; ExternalWritable := 'False'} : Int;
      ldt_MQTT { ExternalAccessible := 'False'; ExternalVisible := 'False'; ExternalWritable := 'False'} : Date_And_Time;
      li_Return_LDT { ExternalAccessible := 'False'; ExternalVisible := 'False'; ExternalWritable := 'False'} : Int;
      lx_Start_TON_Wait { ExternalAccessible := 'False'; ExternalVisible := 'False'; ExternalWritable := 'False'} : Bool;
      ldi_StepHorizontal { ExternalAccessible := 'False'; ExternalVisible := 'False'; ExternalWritable := 'False'} : DInt;
      ldi_StepVertical { ExternalAccessible := 'False'; ExternalVisible := 'False'; ExternalWritable := 'False'} : DInt;
      lfb_TON_Wait {InstructionName := 'TON_TIME'; LibVersion := '1.0'; ExternalAccessible := 'False'; ExternalVisible := 'False'; ExternalWritable := 'False'; S7_SetPoint := 'False'} : TON_TIME;
      lfb_TON_State {InstructionName := 'TON_TIME'; LibVersion := '1.0'; ExternalAccessible := 'False'; ExternalVisible := 'False'; ExternalWritable := 'False'; S7_SetPoint := 'False'} : TON_TIME;
      lfb_F_TRIG_Set_Pos {InstructionName := 'F_TRIG'; LibVersion := '1.0'; ExternalAccessible := 'False'; ExternalVisible := 'False'; ExternalWritable := 'False'; S7_SetPoint := 'False'} : F_TRIG;
   END_VAR


BEGIN
	IF #lx_Init THEN

	    // Restart after set Positioning
	    IF "gtyp_Setup".x_Set_Pos_Activ OR "gtyp_SSC".x_Start_Park_Position THEN
	        #li_StepCase := 0;
	    END_IF;

	    // falling edge Set Pos
	    #lfb_F_TRIG_Set_Pos(CLK:= "gtyp_Setup".x_Set_Pos_Activ);

	    IF #lfb_F_TRIG_Set_Pos.Q THEN
	        #lx_FirstCentre := TRUE;
	    END_IF;

	    #lfb_TON_Wait(IN := #lx_Start_TON_Wait,
	                     PT := #lt_TON_Wait);

	    // wait time state
	    #lfb_TON_State(IN := NOT #lx_Start_TON_State,
	                   PT := T#2s);

	    // state of the ssc cyclically transmitted to the cloud
	    IF #lfb_TON_State.Q AND NOT #lx_Start_TON_State THEN
	        #lx_Start_TON_State := TRUE;
	        #li_Return_LDT := RD_SYS_T(#ldt_MQTT);
	        "gtyp_Interface_Dashboard".Subscribe.PosPanTiltUnit.ldt_ts := DT_TO_LDT(#ldt_MQTT);
	    END_IF;

	    // restart wait time state
	    IF NOT #lfb_TON_State.Q AND #lx_Start_TON_State THEN
	        #lx_Start_TON_State := FALSE;
	    END_IF;

	    CASE #li_StepCase OF

	        0:  // Init
	            #lx_Start_TON_State := FALSE;
	            "gtyp_SSC".Horizontal_Axis.x_Start_Positioning  := FALSE;
	            "gtyp_SSC".Vertical_Axis.x_Start_Positioning    := FALSE;

	            IF NOT "gtyp_Setup".x_Set_Pos_Activ AND NOT "gtyp_SSC".x_Start_Park_Position THEN
	                #li_StepCase := 10;
	            END_IF;

	        10: // Deciding which route to take

	            IF ("gtyp_Interface_Dashboard".Publish.PosPanTiltUnit.ldt_ts > #lldt_ts_old) OR #lx_FirstCentre THEN

	                #lldt_ts_old := "gtyp_Interface_Dashboard".Publish.PosPanTiltUnit.ldt_ts;

	                // convert the degrees to position
	                #ldi_StepHorizontal := REAL_TO_DINT("FC_Scale_linear"(inr_Y1 := DINT_TO_REAL("gtyp_SSC".Horizontal_Axis.Config.di_Neg_Soft_Switch),
	                                                                                                          inr_Y2 := DINT_TO_REAL("gtyp_SSC".Horizontal_Axis.Config.di_Pos_Soft_Switch),
	                                                                                                          inr_X1 := 0.0,
	                                                                                                          inr_X2 := 180.0,
	                                                                                                          inr_X := DINT_TO_REAL("gtyp_Interface_Dashboard".Publish.PosPanTiltUnit.i_degree)));
	                #ldi_StepVertical := REAL_TO_DINT("FC_Scale_linear"(inr_Y1 := DINT_TO_REAL("gtyp_SSC".Vertical_Axis.Config.di_Neg_Soft_Switch),
	                                                                                                      inr_Y2 := DINT_TO_REAL("gtyp_SSC".Vertical_Axis.Config.di_Pos_Soft_Switch),
	                                                                                                      inr_X1 := 0.0,
	                                                                                                      inr_X2 := 180.0,
	                                                                                                      inr_X := DINT_TO_REAL("gtyp_Interface_Dashboard".Publish.PosPanTiltUnit.i_degree)));
	                // Procedure - relmove_left
	                IF ("gtyp_Interface_Dashboard".Publish.PosPanTiltUnit.s_cmd = 'relmove_left')
	                    AND (("gtyp_SSC".Horizontal_Axis.di_Actual_Position - #ldi_StepHorizontal) > "gtyp_SSC".Horizontal_Axis.Config.di_Neg_Soft_Switch + 15)
	                    AND NOT "IX_SSC_RefSwitchHorizontalAxis_I2" THEN
	                    #ldi_TargetPosition_Horizontal := "gtyp_SSC".Horizontal_Axis.di_Actual_Position - #ldi_StepHorizontal;
	                    "gtyp_SSC".Horizontal_Axis.di_Target_Position := #ldi_TargetPosition_Horizontal;
	                    "gtyp_SSC".Horizontal_Axis.x_Start_Positioning := TRUE;
	                    #li_StepCase := 70;
	                // Procedure - relmove_right
	                ELSIF ("gtyp_Interface_Dashboard".Publish.PosPanTiltUnit.s_cmd = 'relmove_right')
	                    AND (("gtyp_SSC".Horizontal_Axis.di_Actual_Position + #ldi_StepHorizontal) < "gtyp_SSC".Horizontal_Axis.Config.di_Pos_Soft_Switch - 15) THEN
	                    #ldi_TargetPosition_Horizontal := "gtyp_SSC".Horizontal_Axis.di_Actual_Position + #ldi_StepHorizontal;
	                    "gtyp_SSC".Horizontal_Axis.di_Target_Position := #ldi_TargetPosition_Horizontal;
	                    "gtyp_SSC".Horizontal_Axis.x_Start_Positioning := TRUE;
	                    #li_StepCase := 70;
	                // Procedure - relmove_up
	                ELSIF ("gtyp_Interface_Dashboard".Publish.PosPanTiltUnit.s_cmd = 'relmove_up')
	                    AND (("gtyp_SSC".Vertical_Axis.di_Actual_Position + #ldi_StepHorizontal) < "gtyp_SSC".Vertical_Axis.Config.di_Pos_Soft_Switch - 15) THEN
	                    #ldi_TargetPosition_Vertical := "gtyp_SSC".Vertical_Axis.di_Actual_Position + #ldi_StepVertical;
	                    "gtyp_SSC".Vertical_Axis.di_Target_Position := #ldi_TargetPosition_Vertical;
	                    "gtyp_SSC".Vertical_Axis.x_Start_Positioning := TRUE;
	                    #li_StepCase := 80;
	                // Procedure - relmove_down
	                ELSIF ("gtyp_Interface_Dashboard".Publish.PosPanTiltUnit.s_cmd = 'relmove_down')
	                    AND (("gtyp_SSC".Vertical_Axis.di_Actual_Position - #ldi_StepVertical) > "gtyp_SSC".Vertical_Axis.Config.di_Neg_Soft_Switch + 15)
	                    AND NOT "IX_SSC_RefSwitchVerticalAxis_I1" THEN
	                    #ldi_TargetPosition_Vertical := "gtyp_SSC".Vertical_Axis.di_Actual_Position - #ldi_StepVertical;
	                    "gtyp_SSC".Vertical_Axis.di_Target_Position := #ldi_TargetPosition_Vertical;
	                    "gtyp_SSC".Vertical_Axis.x_Start_Positioning := TRUE;
	                    #li_StepCase := 80;
	                // Procedure - first
	                ELSIF #lx_FirstCentre THEN
	                    #li_StepCase := 20;
	                // Procedure - home
	                ELSIF ("gtyp_Interface_Dashboard".Publish.PosPanTiltUnit.s_cmd = 'home') THEN
	                    #li_StepCase := 60;
	                // Procedure - start_pan
	                ELSIF ("gtyp_Interface_Dashboard".Publish.PosPanTiltUnit.s_cmd = 'start_pan')
	                    AND ("gtyp_SSC".Horizontal_Axis.di_Actual_Position > "gtyp_SSC".Horizontal_Axis.Config.di_Neg_Soft_Switch + 15)
	                    AND NOT "IX_SSC_RefSwitchHorizontalAxis_I2" THEN
	                    #ldi_TargetPosition_Horizontal := "gtyp_SSC".Horizontal_Axis.Config.di_Neg_Soft_Switch + 15;
	                    "gtyp_SSC".Horizontal_Axis.di_Target_Position := #ldi_TargetPosition_Horizontal;
	                    "gtyp_SSC".Horizontal_Axis.x_Start_Positioning := TRUE;
	                    #li_StepCase := 70;
	                // Procedure - end_pan
	                ELSIF ("gtyp_Interface_Dashboard".Publish.PosPanTiltUnit.s_cmd = 'end_pan')
	                    AND ("gtyp_SSC".Horizontal_Axis.di_Actual_Position < "gtyp_SSC".Horizontal_Axis.Config.di_Pos_Soft_Switch - 15) THEN
	                    #ldi_TargetPosition_Horizontal := "gtyp_SSC".Horizontal_Axis.Config.di_Pos_Soft_Switch - 15;
	                    "gtyp_SSC".Horizontal_Axis.di_Target_Position := #ldi_TargetPosition_Horizontal;
	                    "gtyp_SSC".Horizontal_Axis.x_Start_Positioning := TRUE;
	                    #li_StepCase := 70;
	                // Procedure - start_tilt
	                ELSIF ("gtyp_Interface_Dashboard".Publish.PosPanTiltUnit.s_cmd = 'start_tilt')
	                    AND ("gtyp_SSC".Vertical_Axis.di_Actual_Position > "gtyp_SSC".Vertical_Axis.Config.di_Neg_Soft_Switch + 15)
	                    AND NOT "IX_SSC_RefSwitchVerticalAxis_I1" THEN
	                    #ldi_TargetPosition_Vertical := "gtyp_SSC".Vertical_Axis.Config.di_Neg_Soft_Switch + 15;
	                    "gtyp_SSC".Vertical_Axis.di_Target_Position := #ldi_TargetPosition_Vertical;
	                    "gtyp_SSC".Vertical_Axis.x_Start_Positioning := TRUE;
	                    #li_StepCase := 80;
	                // Procedure - end_tilt
	                ELSIF ("gtyp_Interface_Dashboard".Publish.PosPanTiltUnit.s_cmd = 'end_tilt')
	                    AND ("gtyp_SSC".Vertical_Axis.di_Actual_Position < "gtyp_SSC".Vertical_Axis.Config.di_Pos_Soft_Switch - 15) THEN
	                    #ldi_TargetPosition_Vertical := "gtyp_SSC".Vertical_Axis.Config.di_Pos_Soft_Switch - 15;
	                    "gtyp_SSC".Vertical_Axis.di_Target_Position := #ldi_TargetPosition_Vertical;
	                    "gtyp_SSC".Vertical_Axis.x_Start_Positioning := TRUE;
	                    #li_StepCase := 80;
	                END_IF;
	            END_IF;

	        20: // homing vertical/horizontal axis
	            "gtyp_SSC".Horizontal_Axis.x_Reference  := TRUE;
	            "gtyp_SSC".Vertical_Axis.x_Reference    := TRUE;

	            IF NOT "gtyp_SSC".Horizontal_Axis.x_Referenced AND NOT "gtyp_SSC".Vertical_Axis.x_Referenced THEN
	               #li_StepCase := 30;
	            END_IF;

	        30: // homed vertical/horizontal axis
	            IF "gtyp_SSC".Horizontal_Axis.x_Referenced THEN
	                "gtyp_SSC".Horizontal_Axis.x_Reference := FALSE;
	            END_IF;
	            IF "gtyp_SSC".Vertical_Axis.x_Referenced THEN
	                "gtyp_SSC".Vertical_Axis.x_Reference := FALSE;
	            END_IF;

	            IF "gtyp_SSC".Horizontal_Axis.x_Referenced AND "gtyp_SSC".Vertical_Axis.x_Referenced THEN
	                "gtyp_SSC".Horizontal_Axis.x_Reference := FALSE;
	                "gtyp_SSC".Vertical_Axis.x_Reference := FALSE;
	                #lx_Start_TON_Wait := TRUE;
	                #li_StepCase := 40;
	            END_IF;

	        40: // wait sequence
	            IF #lfb_TON_Wait.Q THEN
	                #lx_Start_TON_Wait := FALSE;
	                #li_StepCase := 50;
	            END_IF;

	        50: // Position horizontal/vertical axis and reached
	            "gtyp_SSC".Horizontal_Axis.di_Target_Position   := "gtyp_SSC".di_Pos_HBW_Horizontal;
	            "gtyp_SSC".Horizontal_Axis.x_Start_Positioning  := TRUE;
	            "gtyp_SSC".Vertical_Axis.di_Target_Position     := "gtyp_SSC".di_Pos_HBW_Vertical;
	            "gtyp_SSC".Vertical_Axis.x_Start_Positioning    := TRUE;

	            IF ("gtyp_SSC".Horizontal_Axis.di_Actual_Position <= ("gtyp_SSC".di_Pos_HBW_Horizontal + "gtyp_SSC".Horizontal_Axis.Config.di_Pos_Window))
	                AND ("gtyp_SSC".Horizontal_Axis.di_Actual_Position >= ("gtyp_SSC".di_Pos_HBW_Horizontal - "gtyp_SSC".Horizontal_Axis.Config.di_Pos_Window))
	                AND "gtyp_SSC".Horizontal_Axis.x_Position_Reached THEN
	                "gtyp_SSC".Horizontal_Axis.x_Start_Positioning := FALSE;
	            END_IF;

	            IF ("gtyp_SSC".Vertical_Axis.di_Actual_Position <= ("gtyp_SSC".di_Pos_HBW_Vertical + "gtyp_SSC".Vertical_Axis.Config.di_Pos_Window))
	                AND ("gtyp_SSC".Vertical_Axis.di_Actual_Position >= ("gtyp_SSC".di_Pos_HBW_Vertical - "gtyp_SSC".Vertical_Axis.Config.di_Pos_Window))
	                AND "gtyp_SSC".Vertical_Axis.x_Position_Reached THEN
	                "gtyp_SSC".Vertical_Axis.x_Start_Positioning := FALSE;
	            END_IF;

	            IF ("gtyp_SSC".Horizontal_Axis.di_Actual_Position <= ("gtyp_SSC".di_Pos_HBW_Horizontal + "gtyp_SSC".Horizontal_Axis.Config.di_Pos_Window))
	                AND ("gtyp_SSC".Horizontal_Axis.di_Actual_Position >= ("gtyp_SSC".di_Pos_HBW_Horizontal - "gtyp_SSC".Horizontal_Axis.Config.di_Pos_Window))
	                AND "gtyp_SSC".Horizontal_Axis.x_Position_Reached
	                AND ("gtyp_SSC".Vertical_Axis.di_Actual_Position <= ("gtyp_SSC".di_Pos_HBW_Vertical + "gtyp_SSC".Vertical_Axis.Config.di_Pos_Window))
	                AND ("gtyp_SSC".Vertical_Axis.di_Actual_Position >= ("gtyp_SSC".di_Pos_HBW_Vertical - "gtyp_SSC".Vertical_Axis.Config.di_Pos_Window))
	                AND "gtyp_SSC".Vertical_Axis.x_Position_Reached THEN
	                "gtyp_SSC".Horizontal_Axis.x_Start_Positioning := FALSE;
	                "gtyp_SSC".Vertical_Axis.x_Start_Positioning := FALSE;
	                #lx_FirstCentre := FALSE;
	                #li_StepCase := 90;
	            END_IF;

	        60: // Position Centre horizontal/vertical axis and reached
	            "gtyp_SSC".Horizontal_Axis.di_Target_Position := "gtyp_SSC".di_Pos_Centre_Horizontal;
	            "gtyp_SSC".Horizontal_Axis.x_Start_Positioning := TRUE;
	            "gtyp_SSC".Vertical_Axis.di_Target_Position := "gtyp_SSC".di_Pos_Centre_Vertical;
	            "gtyp_SSC".Vertical_Axis.x_Start_Positioning := TRUE;

	            IF ("gtyp_SSC".Horizontal_Axis.di_Actual_Position <= ("gtyp_SSC".di_Pos_Centre_Horizontal + "gtyp_SSC".Horizontal_Axis.Config.di_Pos_Window))
	                AND ("gtyp_SSC".Horizontal_Axis.di_Actual_Position >= ("gtyp_SSC".di_Pos_Centre_Horizontal - "gtyp_SSC".Horizontal_Axis.Config.di_Pos_Window))
	                AND "gtyp_SSC".Horizontal_Axis.x_Position_Reached THEN
	                "gtyp_SSC".Horizontal_Axis.x_Start_Positioning := FALSE;
	            END_IF;

	            IF ("gtyp_SSC".Vertical_Axis.di_Actual_Position <= ("gtyp_SSC".di_Pos_Centre_Vertical + "gtyp_SSC".Vertical_Axis.Config.di_Pos_Window))
	                AND ("gtyp_SSC".Vertical_Axis.di_Actual_Position >= ("gtyp_SSC".di_Pos_Centre_Vertical - "gtyp_SSC".Vertical_Axis.Config.di_Pos_Window))
	                AND "gtyp_SSC".Vertical_Axis.x_Position_Reached THEN
	                "gtyp_SSC".Vertical_Axis.x_Start_Positioning := FALSE;
	            END_IF;

	            IF ("gtyp_SSC".Horizontal_Axis.di_Actual_Position <= ("gtyp_SSC".di_Pos_Centre_Horizontal + "gtyp_SSC".Horizontal_Axis.Config.di_Pos_Window))
	                AND ("gtyp_SSC".Horizontal_Axis.di_Actual_Position >= ("gtyp_SSC".di_Pos_Centre_Horizontal - "gtyp_SSC".Horizontal_Axis.Config.di_Pos_Window))
	                AND "gtyp_SSC".Horizontal_Axis.x_Position_Reached
	                AND ("gtyp_SSC".Vertical_Axis.di_Actual_Position <= ("gtyp_SSC".di_Pos_Centre_Vertical + "gtyp_SSC".Vertical_Axis.Config.di_Pos_Window))
	                AND ("gtyp_SSC".Vertical_Axis.di_Actual_Position >= ("gtyp_SSC".di_Pos_Centre_Vertical - "gtyp_SSC".Vertical_Axis.Config.di_Pos_Window))
	                AND "gtyp_SSC".Vertical_Axis.x_Position_Reached THEN
	                "gtyp_SSC".Horizontal_Axis.x_Start_Positioning := FALSE;
	                "gtyp_SSC".Vertical_Axis.x_Start_Positioning := FALSE;
	                #lx_FirstCentre := FALSE;
	                #li_StepCase := 90;
	            END_IF;

	        70: // Position horizontal axis reached
	            IF ("gtyp_SSC".Horizontal_Axis.di_Actual_Position <= (#ldi_TargetPosition_Horizontal + "gtyp_SSC".Horizontal_Axis.Config.di_Pos_Window))
	                AND ("gtyp_SSC".Horizontal_Axis.di_Actual_Position >= (#ldi_TargetPosition_Horizontal - "gtyp_SSC".Horizontal_Axis.Config.di_Pos_Window))
	                AND "gtyp_SSC".Horizontal_Axis.x_Position_Reached THEN
	                "gtyp_SSC".Horizontal_Axis.x_Start_Positioning := FALSE;
	                #li_StepCase := 90;
	            END_IF;

	        80: // Position vertical axis reached
	            IF ("gtyp_SSC".Vertical_Axis.di_Actual_Position <= (#ldi_TargetPosition_Vertical + "gtyp_SSC".Vertical_Axis.Config.di_Pos_Window))
	                AND ("gtyp_SSC".Vertical_Axis.di_Actual_Position >= (#ldi_TargetPosition_Vertical - "gtyp_SSC".Vertical_Axis.Config.di_Pos_Window))
	                AND "gtyp_SSC".Vertical_Axis.x_Position_Reached THEN
	                "gtyp_SSC".Vertical_Axis.x_Start_Positioning := FALSE;
	                #li_StepCase := 90;
	            END_IF;

	        90: // convert the position to degrees
	            "gtyp_Interface_Dashboard".Subscribe.PosPanTiltUnit.r_pan := "FC_Scale_linear"(inr_Y1 := -1.0,
	                                                                                           inr_Y2 := 1.0,
	                                                                                           inr_X1 := DINT_TO_REAL("gtyp_SSC".Horizontal_Axis.Config.di_Neg_Soft_Switch),
	                                                                                           inr_X2 := DINT_TO_REAL("gtyp_SSC".Horizontal_Axis.Config.di_Pos_Soft_Switch),
	                                                                                           inr_X := "gtyp_SSC".Horizontal_Axis.di_Actual_Position);
	            "gtyp_Interface_Dashboard".Subscribe.PosPanTiltUnit.r_tilt:= "FC_Scale_linear"(inr_Y1 := -1.0,
	                                                                                           inr_Y2 := 1.0,
	                                                                                           inr_X1 := DINT_TO_REAL("gtyp_SSC".Vertical_Axis.Config.di_Neg_Soft_Switch),
	                                                                                           inr_X2 := DINT_TO_REAL("gtyp_SSC".Vertical_Axis.Config.di_Pos_Soft_Switch),
	                                                                                           inr_X := "gtyp_SSC".Vertical_Axis.di_Actual_Position);

	            #li_Return_write := RD_SYS_T(#ldt_write);
	            "gtyp_Interface_Dashboard".Subscribe.PosPanTiltUnit.ldt_ts := DT_TO_LDT(#ldt_write);
	            #lx_Start_TON_Wait := TRUE;
	            #li_StepCase := 100;

	        100:// wait sequence
	            IF #lfb_TON_Wait.Q THEN
	                #lx_Start_TON_Wait := FALSE;
	                #li_StepCase := 0;
	            END_IF;
	    // Statement section ELSE
	    ELSE
	        ;
	    END_CASE;

	ELSE
	    #lx_Init := TRUE;
	    #lx_FirstCentre := TRUE;

	    "gtyp_SSC".x_Start_Park_Position := FALSE;
	    "gtyp_SSC".x_Park_Position_Reached := FALSE;
	    "gtyp_SSC".x_Error := FALSE;
	END_IF;
END_FUNCTION_BLOCK

FUNCTION_BLOCK "PRG_SLD_Calibration_Color"
TITLE = Program Calibration Color Sensor SLD
{ S7_Optimized_Access := 'TRUE' }
AUTHOR : 'A.Schaefer'
VERSION : 0.0
   VAR
      lx_Init { ExternalAccessible := 'False'; ExternalVisible := 'False'; ExternalWritable := 'False'} : Bool;
      lx_Start_TON_Wait { ExternalAccessible := 'False'; ExternalVisible := 'False'; ExternalWritable := 'False'} : Bool;
      lx_Start_Positioning_m { ExternalAccessible := 'False'; ExternalVisible := 'False'; ExternalWritable := 'False'} : Bool;
      lt_TON_Wait { ExternalAccessible := 'False'; ExternalVisible := 'False'; ExternalWritable := 'False'} : Time;
      li_StepCase { ExternalAccessible := 'False'; ExternalVisible := 'False'; ExternalWritable := 'False'} : Int;
      lw_ColorValueMin { ExternalAccessible := 'False'; ExternalVisible := 'False'; ExternalWritable := 'False'} : Word;
      ldi_Pos_Horizontal { ExternalAccessible := 'False'; ExternalVisible := 'False'; ExternalWritable := 'False'} : DInt;
      ldi_Pos_Vertical { ExternalAccessible := 'False'; ExternalVisible := 'False'; ExternalWritable := 'False'} : DInt;
      lfb_R_Trig_Deaktivate {InstructionName := 'R_TRIG'; LibVersion := '1.0'; ExternalAccessible := 'False'; ExternalVisible := 'False'; ExternalWritable := 'False'; S7_SetPoint := 'False'} : R_TRIG;
      lfb_TON_Wait {InstructionName := 'TON_TIME'; LibVersion := '1.0'; ExternalAccessible := 'False'; ExternalVisible := 'False'; ExternalWritable := 'False'; S7_SetPoint := 'False'} : TON_TIME;
   END_VAR


BEGIN
	IF #lx_Init THEN

	    // FB TON Wait
	    #lfb_TON_Wait(IN := #lx_Start_TON_Wait,
	                  PT := #lt_TON_Wait);

	    #lfb_R_Trig_Deaktivate(CLK:= NOT "gtyp_Setup".x_Color_Sensor_Calibration
	                           OR NOT ("gtyp_Setup".i_Color_Sensor_Selection = 2));
	    // Deaktivate step 0
	    IF #lfb_R_Trig_Deaktivate.Q THEN
	        "gtyp_Setup".x_Calculate_Value_Color := FALSE;
	        "gtyp_Setup".x_Set_Calib_Value_Color_Blue := FALSE;
	        "gtyp_Setup".x_Set_Calib_Value_Color_Red := FALSE;
	        "gtyp_Setup".x_Set_Calib_Value_Color_White := FALSE;
	        "gtyp_Setup".w_Calib_ColorValue_Blue := 0;
	        "gtyp_Setup".w_Calib_ColorValue_Red := 0;
	        "gtyp_Setup".w_Calib_ColorValue_White := 0;
	        "gtyp_Setup".w_Threshold_Red_Blue := 0;
	        "gtyp_Setup".w_Threshold_White_Red := 0;
	        "QX_SLD_M1_ConveyorBelt_Q1" := FALSE;
	        #lw_ColorValueMin := 16#FF;
	        #li_StepCase            := 0;
	    END_IF;

	    // step chain HBW
	    CASE #li_StepCase OF

	        0:  // init
	            #lx_Start_TON_Wait := FALSE;
	            #li_StepCase := 10;

	        10:  // Set Calibration activ?
	            IF "gtyp_Setup".x_Color_Sensor_Calibration
	                AND ("gtyp_Setup".i_Color_Sensor_Selection = 2) THEN
	                "gtyp_Setup".x_Calculate_Value_Color := FALSE;
	                "gtyp_Setup".x_Set_Calib_Value_Color_Blue := FALSE;
	                "gtyp_Setup".x_Set_Calib_Value_Color_Red := FALSE;
	                "gtyp_Setup".x_Set_Calib_Value_Color_White := FALSE;
	                "gtyp_Setup".w_Calib_ColorValue_Blue := 0;
	                "gtyp_Setup".w_Calib_ColorValue_Red := 0;
	                "gtyp_Setup".w_Calib_ColorValue_White := 0;
	                "gtyp_Setup".w_Threshold_Red_Blue := 0;
	                "gtyp_Setup".w_Threshold_White_Red := 0;
	                "QX_SLD_M1_ConveyorBelt_Q1" := FALSE;
	                #lw_ColorValueMin := 16#FFFF;
	                #li_StepCase := 20;
	            END_IF;

	        20: // wait for set Values or Calculate

	            IF NOT "IX_SLD_LightBarrierInlet_I2" THEN
	                "QX_SLD_M1_ConveyorBelt_Q1" := TRUE;
	                #lw_ColorValueMin := 16#FFFF;
	            END_IF;

	            IF #lw_ColorValueMin > "IW_SLD_ColorSensor_A4" THEN
	                #lw_ColorValueMin := "IW_SLD_ColorSensor_A4";
	            END_IF;

	            IF NOT "IX_SLD_LightBarrierBehindColorSensor_I3" THEN
	                "QX_SLD_M1_ConveyorBelt_Q1" := FALSE;
	            END_IF;

	            // Start new Positioning
	            IF "gtyp_Setup".x_Set_Calib_Value_Color_Blue THEN
	                "gtyp_Setup".w_Calib_ColorValue_Blue := #lw_ColorValueMin;
	                "gtyp_Setup".x_Set_Calib_Value_Color_Blue := FALSE;
	            ELSIF "gtyp_Setup".x_Set_Calib_Value_Color_Red THEN
	                "gtyp_Setup".w_Calib_ColorValue_Red := #lw_ColorValueMin;
	                "gtyp_Setup".x_Set_Calib_Value_Color_Red := FALSE;
	            ELSIF "gtyp_Setup".x_Set_Calib_Value_Color_White THEN
	                "gtyp_Setup".w_Calib_ColorValue_White := #lw_ColorValueMin;
	                "gtyp_Setup".x_Set_Calib_Value_Color_White := FALSE;
	            END_IF;

	            "gtyp_Setup".w_Threshold_White_Red := "gtyp_Setup".w_Calib_ColorValue_White + (("gtyp_Setup".w_Calib_ColorValue_Red - "gtyp_Setup".w_Calib_ColorValue_White) / 2);
	            "gtyp_Setup".w_Threshold_Red_Blue := "gtyp_Setup".w_Calib_ColorValue_Red + (("gtyp_Setup".w_Calib_ColorValue_Blue - "gtyp_Setup".w_Calib_ColorValue_Red) / 2);

	            IF "gtyp_Setup".x_Calculate_Value_Color THEN
	                "gtyp_SLD".w_Threshold_White_Red := "gtyp_Setup".w_Threshold_White_Red;
	                "gtyp_SLD".w_Threshold_Red_Blue := "gtyp_Setup".w_Threshold_Red_Blue;
	                "gtyp_Setup".x_Calculate_Value_Color := FALSE;
	            END_IF;

	            // Statement section ELSE
	        ELSE
	            ;
	    END_CASE;

	    IF ("gtyp_Setup".i_Color_Sensor_Selection = 2) THEN
	        // Reload Pos Value
	        "gtyp_Setup".w_Actual_ColorValue := "IW_SLD_ColorSensor_A4";
	    END_IF;
	ELSE
	    #lx_Init := TRUE;
	END_IF;
END_FUNCTION_BLOCK

FUNCTION_BLOCK "PRG_SSC_Axis_Vertical"
TITLE = Program Axis vertical SSC
{ S7_Optimized_Access := 'TRUE' }
AUTHOR : 'A.Schaefer'
VERSION : 0.0
   VAR
      lx_Init { ExternalAccessible := 'False'; ExternalVisible := 'False'; ExternalWritable := 'False'} : Bool;
      lfb_Vertical_Axis { ExternalAccessible := 'False'; ExternalVisible := 'False'; ExternalWritable := 'False'; S7_SetPoint := 'False'} : "FB_Axis";
   END_VAR


BEGIN
	IF #lx_Init THEN

	    // FB Axis vertical
	    #lfb_Vertical_Axis( ini_Axis                := 5,
	                        indi_Increment          := "gtyp_SSC".Vertical_Axis.di_Increment,
	                        inx_Ref_Switch          := "IX_SSC_RefSwitchVerticalAxis_I1",
	                        inx_Referencing         := "gtyp_SSC".Vertical_Axis.x_Reference,
	                        inx_Start_Positioning   := "gtyp_SSC".Vertical_Axis.x_Start_Positioning,
	                        indi_Target_Position    := "gtyp_SSC".Vertical_Axis.di_Target_Position,
	                        ini_PWM               := "gtyp_SSC".Vertical_Axis.i_PWM,
	                        inouttyp_Config         := "gtyp_SSC".Vertical_Axis.Config,
	                        inouttyp_Setup          := "gtyp_SetupAxis");

	    "QX_SSC_M1_VerticalAxisUp_Q1"                    := #lfb_Vertical_Axis.outx_Motor_Pos;
	    "QX_SSC_M1_VerticalAxisDown_Q2"                  := #lfb_Vertical_Axis.outx_Motor_Neg;
	    "QW_SSC_PWM_Vertical_M1"                         := #lfb_Vertical_Axis.outi_Motor_PWM;
	    "gtyp_SSC".Vertical_Axis.di_Actual_Position   := #lfb_Vertical_Axis.outdi_Actual_Position;
	    "gtyp_SSC".Vertical_Axis.x_Referenced         := #lfb_Vertical_Axis.outx_Referenced;
	    "gtyp_SSC".Vertical_Axis.x_Position_Reached   := #lfb_Vertical_Axis.outx_Position_Reached;
	ELSE
	    #lx_Init := TRUE;
	END_IF;
END_FUNCTION_BLOCK

FUNCTION_BLOCK "PRG_SSC_Set_Park_Position"
TITLE = Program Set Positioning SSC
{ S7_Optimized_Access := 'TRUE' }
AUTHOR : 'A.Schaefer'
VERSION : 0.0
   VAR
      lx_Init { ExternalAccessible := 'False'; ExternalVisible := 'False'; ExternalWritable := 'False'} : Bool;
      lx_Start_TON_Wait { ExternalAccessible := 'False'; ExternalVisible := 'False'; ExternalWritable := 'False'} : Bool;
      lt_TON_Wait { ExternalAccessible := 'False'; ExternalVisible := 'False'; ExternalWritable := 'False'} : Time;
      li_StepCase { ExternalAccessible := 'False'; ExternalVisible := 'False'; ExternalWritable := 'False'} : Int;
      lfb_TON_Wait {InstructionName := 'TON_TIME'; LibVersion := '1.0'; ExternalAccessible := 'False'; ExternalVisible := 'False'; ExternalWritable := 'False'; S7_SetPoint := 'False'} : TON_TIME;
      lfb_R_Trig_Start_Park_Pos {InstructionName := 'R_TRIG'; LibVersion := '1.0'; ExternalAccessible := 'False'; ExternalVisible := 'False'; ExternalWritable := 'False'; S7_SetPoint := 'False'} : R_TRIG;
   END_VAR


BEGIN
	IF #lx_Init THEN

	    // FB TON Wait
	    #lfb_TON_Wait(IN := #lx_Start_TON_Wait,
	                  PT := #lt_TON_Wait);

	    #lfb_R_Trig_Start_Park_Pos(CLK := "gtyp_Setup".x_Park_Position
	                               OR "IX_Set_Park_Position");

	    // Set Start Park Position
	    IF #lfb_R_Trig_Start_Park_Pos.Q THEN
	        "gtyp_SSC".x_Start_Park_Position := TRUE;
	        #li_StepCase := 0;
	    END_IF;

	    // not Start Park Pos Step 0
	    IF NOT "gtyp_SSC".x_Start_Park_Position THEN
	        #li_StepCase := 0;
	    END_IF;

	    // step chain HBW
	    CASE #li_StepCase OF

	        0:  // init
	            #lx_Start_TON_Wait := FALSE;
	            #li_StepCase := 10;

	        10:  // Set Positioning activ?
	            IF "gtyp_SSC".x_Start_Park_Position AND NOT "gtyp_SSC".x_Park_Position_Reached THEN
	                "gtyp_SSC".Horizontal_Axis.x_Start_Positioning := FALSE;
	                "gtyp_SSC".Vertical_Axis.x_Start_Positioning := FALSE;
	                "gtyp_SSC".Horizontal_Axis.x_Reference := FALSE;
	                "gtyp_SSC".Vertical_Axis.x_Reference := FALSE;
	                 #li_StepCase := 20;
	            END_IF;

	        20: // homing vertical axis
	            "gtyp_SSC".Vertical_Axis.x_Reference := TRUE;

	            IF NOT "gtyp_SSC".Vertical_Axis.x_Referenced THEN
	                #li_StepCase := 30;
	            END_IF;

	        30: // homed vertical axis
	            IF "gtyp_SSC".Vertical_Axis.x_Referenced THEN
	                "gtyp_SSC".Vertical_Axis.x_Reference := FALSE;
	                #li_StepCase := 40;
	            END_IF;

	        40: // homing horizontal axis
	            "gtyp_SSC".Horizontal_Axis.x_Reference := TRUE;

	            IF NOT "gtyp_SSC".Horizontal_Axis.x_Referenced THEN
	                #li_StepCase := 50;
	            END_IF;

	        50: // homed horizontal axis
	            IF "gtyp_SSC".Horizontal_Axis.x_Referenced THEN
	                "gtyp_SSC".Horizontal_Axis.x_Reference := FALSE;
	                #li_StepCase := 60;
	            END_IF;

	        60: // Position horizontal Axis
	            "gtyp_SSC".Horizontal_Axis.di_Target_Position := "gtyp_SSC".di_Pos_Park_Horizontal;
	            "gtyp_SSC".Horizontal_Axis.x_Start_Positioning := TRUE;

	            IF ("gtyp_SSC".Horizontal_Axis.di_Actual_Position <= ("gtyp_SSC".di_Pos_Park_Horizontal + "gtyp_SSC".Horizontal_Axis.Config.di_Pos_Window))
	                AND ("gtyp_SSC".Horizontal_Axis.di_Actual_Position >= ("gtyp_SSC".di_Pos_Park_Horizontal - "gtyp_SSC".Horizontal_Axis.Config.di_Pos_Window))
	                AND "gtyp_SSC".Horizontal_Axis.x_Position_Reached THEN
	                "gtyp_SSC".Horizontal_Axis.x_Start_Positioning := FALSE;
	                #li_StepCase := 70;
	            END_IF;

